C01815=1097.718,-43.728,-51.069,175.704,14.690,152.016
C01816=1097.724,-43.478,-51.082,175.706,14.691,152.016
C01817=1097.729,-43.229,-51.094,175.708,14.691,152.015
C01818=1097.736,-42.979,-51.106,175.710,14.692,152.015
C01819=1097.742,-42.730,-51.119,175.711,14.692,152.015
C01820=1097.748,-42.480,-51.130,175.713,14.693,152.015
C01821=1097.754,-42.230,-51.142,175.715,14.694,152.014
C01822=1097.759,-41.981,-51.154,175.717,14.695,152.014
C01823=1097.766,-41.731,-51.166,175.718,14.695,152.014
C01824=1097.771,-41.482,-51.179,175.720,14.696,152.014
C01825=1097.776,-41.232,-51.190,175.722,14.697,152.013
C01826=1097.783,-40.982,-51.202,175.724,14.697,152.013
C01827=1097.789,-40.732,-51.215,175.726,14.698,152.013
C01828=1097.795,-40.483,-51.226,175.728,14.699,152.012
C01829=1097.801,-40.234,-51.239,175.730,14.700,152.012
C01830=1097.807,-39.984,-51.252,175.732,14.700,152.012
C01831=1097.813,-39.735,-51.263,175.733,14.701,152.012
C01832=1097.819,-39.484,-51.275,175.735,14.702,152.011
C01833=1097.824,-39.234,-51.287,175.737,14.703,152.011
C01834=1097.831,-38.985,-51.299,175.739,14.703,152.011
C01835=1097.836,-38.736,-51.312,175.741,14.704,152.011
C01836=1097.842,-38.486,-51.324,175.743,14.705,152.010
C01837=1097.848,-38.236,-51.337,175.745,14.706,152.010
C01838=1097.854,-37.987,-51.348,175.747,14.706,152.010
C01839=1097.860,-37.737,-51.361,175.748,14.707,152.010
C01840=1097.866,-37.487,-51.373,175.750,14.708,152.009
C01841=1097.871,-37.238,-51.386,175.752,14.709,152.009
C01842=1097.877,-36.988,-51.397,175.754,14.709,152.009
C01843=1097.884,-36.738,-51.409,175.756,14.710,152.009
C01844=1097.889,-36.489,-51.422,175.758,14.711,152.008
C01845=1097.895,-36.239,-51.434,175.760,14.712,152.008
C01846=1097.901,-35.989,-51.447,175.762,14.712,152.008
C01847=1097.906,-35.740,-51.459,175.763,14.713,152.008
C01848=1097.912,-35.490,-51.471,175.765,14.714,152.007
C01849=1097.919,-35.240,-51.483,175.767,14.715,152.007
C01850=1097.924,-34.991,-51.496,175.769,14.715,152.007
C01851=1097.930,-34.741,-51.508,175.771,14.716,152.006
C01852=1097.936,-34.491,-51.521,175.773,14.717,152.006
C01853=1097.941,-34.242,-51.533,175.775,14.717,152.006
C01854=1097.947,-33.992,-51.545,175.777,14.718,152.006
C01855=1097.954,-33.743,-51.557,175.778,14.719,152.005
C01856=1097.960,-33.493,-51.570,175.780,14.720,152.005
C01857=1097.965,-33.244,-51.582,175.782,14.720,152.005
C01858=1097.971,-32.994,-51.595,175.784,14.721,152.005
C01859=1097.977,-32.727,-51.608,175.786,14.722,152.004
C01860=1097.984,-32.460,-51.622,175.788,14.723,152.004
C01861=1097.990,-32.192,-51.635,175.790,14.723,152.004
C01862=1097.996,-31.924,-51.648,175.792,14.725,152.004
C01863=1098.002,-31.674,-51.661,175.794,14.726,152.003
C01864=1098.008,-31.425,-51.673,175.796,14.726,152.003
C01865=1098.013,-31.175,-51.686,175.798,14.727,152.003
C01866=1098.020,-30.926,-51.698,175.800,14.728,152.003
C01867=1098.026,-30.677,-51.711,175.802,14.728,152.002
C01868=1098.032,-30.427,-51.723,175.804,14.729,152.002
C01869=1098.037,-30.178,-51.736,175.806,14.730,152.002
C01870=1098.043,-29.928,-51.748,175.807,14.731,152.001
C01871=1098.049,-29.678,-51.761,175.809,14.731,152.001
C01872=1098.055,-29.428,-51.773,175.812,14.732,152.001
C01873=1098.061,-29.178,-51.786,175.813,14.732,152.001
C01874=1098.066,-28.929,-51.799,175.815,14.733,152.000
C01875=1098.072,-28.680,-51.811,175.817,14.734,152.000
C01876=1098.078,-28.430,-51.824,175.819,14.735,152.000
C01877=1098.085,-28.180,-51.836,175.821,14.735,152.000
C01878=1098.091,-27.930,-51.848,175.823,14.736,151.999
C01879=1098.097,-27.681,-51.862,175.825,14.737,151.999
C01880=1098.102,-27.432,-51.874,175.827,14.738,151.999
C01881=1098.108,-27.182,-51.886,175.828,14.738,151.998
C01882=1098.114,-26.932,-51.899,175.830,14.739,151.998
C01883=1098.120,-26.682,-51.911,175.832,14.740,151.998
C01884=1098.126,-26.433,-51.925,175.834,14.741,151.998
C01885=1098.132,-26.184,-51.937,175.836,14.741,151.997
C01886=1098.137,-25.933,-51.950,175.838,14.742,151.997
C01887=1098.143,-25.684,-51.963,175.840,14.743,151.997
C01888=1098.149,-25.434,-51.976,175.842,14.744,151.997
C01889=1098.155,-25.184,-51.988,175.843,14.744,151.996
C01890=1098.160,-24.935,-52.001,175.845,14.745,151.996
C01891=1098.166,-24.685,-52.013,175.847,14.746,151.996
C01892=1098.172,-24.436,-52.026,175.850,14.747,151.996
C01893=1098.178,-24.186,-52.039,175.852,14.748,151.995
C01894=1098.184,-23.936,-52.052,175.854,14.749,151.995
C01895=1098.190,-23.688,-52.064,175.855,14.749,151.995
C01896=1098.195,-23.438,-52.078,175.857,14.750,151.995
C01897=1098.201,-23.188,-52.090,175.859,14.751,151.994
C01898=1098.207,-22.938,-52.103,175.861,14.752,151.994
C01899=1098.213,-22.689,-52.116,175.863,14.752,151.994
C01900=1098.219,-22.439,-52.129,175.865,14.753,151.993
C01901=1098.225,-22.189,-52.142,175.867,14.754,151.993
C01902=1098.230,-21.940,-52.154,175.869,14.755,151.993
C01903=1098.235,-21.690,-52.167,175.870,14.755,151.993
C01904=1098.242,-21.441,-52.180,175.872,14.756,151.992
C01905=1098.247,-21.191,-52.193,175.875,14.756,151.992
C01906=1098.254,-20.942,-52.206,175.876,14.757,151.992
C01907=1098.260,-20.692,-52.219,175.878,14.758,151.992
C01908=1098.266,-20.442,-52.231,175.881,14.759,151.991
C01909=1098.272,-20.193,-52.245,175.883,14.760,151.991
C01910=1098.276,-19.943,-52.257,175.885,14.761,151.991
C01911=1098.283,-19.694,-52.271,175.887,14.761,151.990
C01912=1098.288,-19.444,-52.283,175.888,14.762,151.990
C01913=1098.294,-19.194,-52.296,175.890,14.763,151.990
C01914=1098.301,-18.945,-52.309,175.892,14.764,151.990
C01915=1098.306,-18.695,-52.322,175.894,14.764,151.989
C01916=1098.312,-18.445,-52.336,175.896,14.765,151.989
C01917=1098.318,-18.195,-52.348,175.898,14.766,151.989
C01918=1098.324,-17.946,-52.361,175.900,14.767,151.989
C01919=1098.330,-17.696,-52.374,175.902,14.767,151.988
C01920=1098.335,-17.447,-52.388,175.904,14.768,151.988
C01921=1098.341,-17.197,-52.400,175.906,14.769,151.988
C01922=1098.347,-16.948,-52.413,175.908,14.770,151.987
C01923=1098.353,-16.680,-52.427,175.910,14.771,151.987
C01924=1098.359,-16.411,-52.441,175.912,14.771,151.987
C01925=1098.366,-16.143,-52.455,175.914,14.772,151.987
C01926=1098.373,-15.875,-52.469,175.917,14.773,151.986
C01927=1098.378,-15.625,-52.483,175.919,14.774,151.986
C01928=1098.384,-15.376,-52.496,175.921,14.774,151.986
C01929=1098.390,-15.126,-52.508,175.923,14.775,151.985
C01930=1098.397,-14.877,-52.522,175.924,14.776,151.985
C01931=1098.402,-14.626,-52.535,175.926,14.777,151.985
C01932=1098.408,-14.377,-52.548,175.928,14.777,151.985
C01933=1098.413,-14.128,-52.561,175.930,14.778,151.984
C01934=1098.419,-13.878,-52.574,175.932,14.779,151.984
C01935=1098.425,-13.629,-52.587,175.934,14.780,151.984
C01936=1098.430,-13.379,-52.601,175.936,14.781,151.984
C01937=1098.436,-13.130,-52.614,175.938,14.782,151.983
C01938=1098.441,-12.880,-52.627,175.940,14.783,151.983
C01939=1098.448,-12.630,-52.640,175.942,14.783,151.983
C01940=1098.454,-12.381,-52.654,175.944,14.784,151.982
C01941=1098.459,-12.131,-52.667,175.946,14.784,151.982
C01942=1098.465,-11.882,-52.680,175.948,14.785,151.982
C01943=1098.471,-11.632,-52.694,175.950,14.786,151.982
C01944=1098.477,-11.382,-52.706,175.952,14.787,151.981
C01945=1098.483,-11.133,-52.720,175.954,14.787,151.981
C01946=1098.488,-10.883,-52.734,175.956,14.789,151.981
C01947=1098.494,-10.633,-52.746,175.958,14.789,151.980
C01948=1098.500,-10.384,-52.760,175.960,14.790,151.980
C01949=1098.506,-10.135,-52.773,175.962,14.790,151.980
C01950=1098.511,-9.884,-52.786,175.964,14.791,151.980
C01951=1098.517,-9.635,-52.800,175.966,14.792,151.979
C01952=1098.524,-9.386,-52.813,175.968,14.793,151.979
C01953=1098.529,-9.136,-52.827,175.970,14.793,151.979
C01954=1098.535,-8.886,-52.839,175.972,14.795,151.978
C01955=1098.540,-8.637,-52.853,175.974,14.796,151.978
C01956=1098.547,-8.387,-52.866,175.976,14.796,151.978
C01957=1098.552,-8.138,-52.880,175.978,14.797,151.978
C01958=1098.558,-7.888,-52.893,175.980,14.797,151.977
C01959=1098.564,-7.638,-52.907,175.982,14.798,151.977
C01960=1098.570,-7.389,-52.920,175.984,14.799,151.977
C01961=1098.575,-7.140,-52.934,175.986,14.800,151.977
C01962=1098.581,-6.890,-52.947,175.989,14.801,151.976
C01963=1098.587,-6.640,-52.960,175.990,14.802,151.976
C01964=1098.593,-6.391,-52.974,175.993,14.802,151.976
C01965=1098.600,-6.141,-52.987,175.994,14.803,151.975
C01966=1098.605,-5.891,-53.001,175.996,14.803,151.975
C01967=1098.611,-5.642,-53.014,175.998,14.804,151.975
C01968=1098.617,-5.393,-53.028,176.000,14.805,151.975
C01969=1098.623,-5.143,-53.041,176.002,14.805,151.974
C01970=1098.628,-4.893,-53.055,176.005,14.807,151.974
C01971=1098.634,-4.643,-53.069,176.007,14.807,151.974
C01972=1098.640,-4.394,-53.082,176.009,14.808,151.973
C01973=1098.645,-4.145,-53.096,176.011,14.809,151.973
C01974=1098.652,-3.895,-53.109,176.012,14.810,151.973
C01975=1098.657,-3.646,-53.123,176.015,14.810,151.972
C01976=1098.664,-3.396,-53.136,176.017,14.811,151.972
C01977=1098.669,-3.146,-53.150,176.018,14.811,151.972
C01978=1098.676,-2.897,-53.164,176.021,14.813,151.972
C01979=1098.681,-2.647,-53.177,176.023,14.813,151.971
C01980=1098.686,-2.397,-53.191,176.025,14.814,151.971
C01981=1098.692,-2.148,-53.204,176.027,14.814,151.971
C01982=1098.698,-1.898,-53.218,176.029,14.815,151.970
C01983=1098.703,-1.649,-53.232,176.031,14.816,151.970
C01984=1098.709,-1.399,-53.245,176.033,14.817,151.970
C01985=1098.715,-1.150,-53.259,176.035,14.818,151.970
C01986=1098.721,-0.900,-53.273,176.037,14.819,151.969
C01987=1098.726,-0.630,-53.287,176.039,14.820,151.969
C01988=1098.733,-0.360,-53.302,176.042,14.820,151.969
C01989=1098.739,-0.091,-53.318,176.044,14.821,151.968
C01990=1098.745,0.179,-53.332,176.046,14.822,151.968
C01991=1098.751,0.429,-53.346,176.048,14.823,151.968
C01992=1098.756,0.678,-53.360,176.051,14.824,151.967
C01993=1098.762,0.927,-53.373,176.052,14.824,151.967
C01994=1098.769,1.178,-53.387,176.054,14.825,151.967
C01995=1098.774,1.427,-53.401,176.056,14.826,151.967
C01996=1098.779,1.677,-53.415,176.058,14.827,151.966
C01997=1098.786,1.926,-53.428,176.060,14.827,151.966
C01998=1098.791,2.176,-53.442,176.063,14.828,151.966
C01999=1098.797,2.425,-53.456,176.065,14.829,151.965
C02000=1098.802,2.675,-53.470,176.067,14.830,151.965
C02001=1098.808,2.924,-53.484,176.069,14.830,151.965
C02002=1098.814,3.174,-53.498,176.071,14.831,151.964
C02003=1098.820,3.423,-53.512,176.073,14.832,151.964
C02004=1098.826,3.673,-53.526,176.075,14.833,151.964
C02005=1098.831,3.922,-53.540,176.077,14.834,151.964
C02006=1098.837,4.172,-53.554,176.079,14.834,151.963
C02007=1098.843,4.421,-53.567,176.081,14.835,151.963
C02008=1098.849,4.672,-53.581,176.083,14.835,151.963
C02009=1098.854,4.921,-53.595,176.085,14.836,151.962
C02010=1098.860,5.170,-53.610,176.088,14.838,151.962
C02011=1098.866,5.420,-53.624,176.090,14.838,151.962
C02012=1098.872,5.669,-53.637,176.092,14.839,151.961
C02013=1098.878,5.919,-53.651,176.094,14.839,151.961
C02014=1098.883,6.169,-53.665,176.096,14.840,151.961
C02015=1098.889,6.418,-53.679,176.098,14.840,151.961
C02016=1098.895,6.667,-53.693,176.100,14.842,151.960
C02017=1098.900,6.917,-53.707,176.102,14.842,151.960
C02018=1098.907,7.167,-53.721,176.104,14.843,151.960
C02019=1098.912,7.416,-53.735,176.106,14.844,151.959
C02020=1098.918,7.665,-53.749,176.108,14.844,151.959
C02021=1098.924,7.915,-53.763,176.111,14.845,151.959
C02022=1098.930,8.165,-53.777,176.113,14.846,151.958
C02023=1098.935,8.415,-53.791,176.115,14.847,151.958
C02024=1098.941,8.664,-53.806,176.117,14.847,151.958
C02025=1098.947,8.913,-53.819,176.119,14.848,151.957
C02026=1098.953,9.163,-53.833,176.122,14.849,151.957
C02027=1098.959,9.412,-53.848,176.123,14.850,151.957
C02028=1098.965,9.662,-53.862,176.126,14.850,151.956
C02029=1098.970,9.911,-53.876,176.127,14.851,151.956
C02030=1098.976,10.161,-53.891,176.129,14.852,151.956
C02031=1098.982,10.411,-53.904,176.132,14.852,151.956
C02032=1098.987,10.660,-53.918,176.134,14.853,151.955
C02033=1098.994,10.910,-53.933,176.136,14.854,151.955
C02034=1098.999,11.159,-53.947,176.138,14.854,151.955
C02035=1099.005,11.409,-53.960,176.140,14.855,151.954
C02036=1099.012,11.658,-53.975,176.142,14.855,151.954
C02037=1099.017,11.908,-53.989,176.145,14.857,151.954
C02038=1099.023,12.158,-54.003,176.147,14.857,151.953
C02039=1099.029,12.407,-54.018,176.149,14.858,151.953
C02040=1099.035,12.657,-54.032,176.151,14.858,151.953
C02041=1099.040,12.906,-54.046,176.153,14.859,151.952
C02042=1099.046,13.155,-54.060,176.156,14.860,151.952
C02043=1099.052,13.405,-54.075,176.158,14.861,151.952
C02044=1099.058,13.655,-54.089,176.160,14.861,151.951
C02045=1099.064,13.905,-54.103,176.162,14.862,151.951
C02046=1099.070,14.154,-54.118,176.164,14.862,151.951
C02047=1099.075,14.403,-54.132,176.167,14.864,151.950
C02048=1099.081,14.652,-54.146,176.168,14.864,151.950
C02049=1099.087,14.903,-54.161,176.171,14.865,151.950
C02050=1099.093,15.152,-54.175,176.173,14.865,151.949
C02051=1099.099,15.424,-54.190,176.175,14.866,151.949
C02052=1099.105,15.695,-54.206,176.177,14.867,151.949
C02053=1099.111,15.968,-54.222,176.180,14.868,151.948
C02054=1099.118,16.239,-54.238,176.182,14.869,151.948
C02055=1099.123,16.489,-54.252,176.184,14.869,151.948
C02056=1099.130,16.738,-54.266,176.186,14.870,151.947
C02057=1099.135,16.987,-54.281,176.189,14.871,151.947
C02058=1099.140,17.237,-54.296,176.191,14.871,151.947
C02059=1099.147,17.487,-54.310,176.193,14.872,151.946
C02060=1099.152,17.736,-54.324,176.195,14.873,151.946
C02061=1099.158,17.985,-54.339,176.198,14.874,151.946
C02062=1099.164,18.236,-54.353,176.200,14.875,151.945
C02063=1099.170,18.485,-54.368,176.202,14.875,151.945
C02064=1099.176,18.734,-54.383,176.204,14.876,151.945
C02065=1099.181,18.984,-54.397,176.206,14.876,151.944
C02066=1099.187,19.233,-54.412,176.209,14.877,151.944
C02067=1099.193,19.483,-54.426,176.210,14.878,151.944
C02068=1099.198,19.732,-54.441,176.213,14.878,151.943
C02069=1099.205,19.982,-54.455,176.215,14.879,151.943
C02070=1099.210,20.232,-54.469,176.218,14.880,151.943
C02071=1099.215,20.481,-54.484,176.219,14.881,151.942
C02072=1099.222,20.730,-54.499,176.222,14.881,151.942
C02073=1099.227,20.980,-54.513,176.223,14.882,151.942
C02074=1099.233,21.229,-54.528,176.226,14.883,151.941
C02075=1099.239,21.479,-54.543,176.228,14.883,151.941
C02076=1099.244,21.729,-54.557,176.230,14.884,151.941
C02077=1099.251,21.978,-54.572,176.232,14.884,151.940
C02078=1099.256,22.227,-54.587,176.234,14.885,151.940
C02079=1099.261,22.477,-54.601,176.237,14.886,151.940
C02080=1099.267,22.727,-54.616,176.239,14.887,151.939
C02081=1099.273,22.976,-54.631,176.241,14.887,151.939
C02082=1099.279,23.226,-54.645,176.243,14.888,151.939
C02083=1099.284,23.475,-54.660,176.246,14.889,151.938
C02084=1099.290,23.724,-54.675,176.248,14.890,151.938
C02085=1099.296,23.974,-54.690,176.250,14.890,151.938
C02086=1099.301,24.224,-54.704,176.252,14.891,151.937
C02087=1099.308,24.473,-54.719,176.255,14.891,151.937
C02088=1099.313,24.722,-54.734,176.257,14.892,151.937
C02089=1099.320,24.972,-54.749,176.259,14.893,151.936
C02090=1099.325,25.221,-54.764,176.261,14.893,151.936
C02091=1099.331,25.472,-54.778,176.264,14.894,151.935
C02092=1099.337,25.720,-54.793,176.266,14.894,151.935
C02093=1099.342,25.970,-54.808,176.268,14.895,151.935
C02094=1099.348,26.219,-54.823,176.270,14.896,151.934
C02095=1099.354,26.469,-54.838,176.273,14.897,151.934
C02096=1099.360,26.718,-54.853,176.275,14.897,151.934
C02097=1099.365,26.968,-54.867,176.277,14.898,151.933
C02098=1099.371,27.218,-54.882,176.279,14.898,151.933
C02099=1099.376,27.467,-54.897,176.282,14.900,151.933
C02100=1099.383,27.716,-54.912,176.284,14.900,151.932
C02101=1099.388,27.966,-54.927,176.286,14.900,151.932
C02102=1099.394,28.215,-54.942,176.288,14.901,151.932
C02103=1099.400,28.464,-54.957,176.291,14.902,151.931
C02104=1099.406,28.714,-54.972,176.293,14.903,151.931
C02105=1099.411,28.963,-54.987,176.295,14.903,151.931
C02106=1099.417,29.213,-55.002,176.298,14.904,151.930
C02107=1099.423,29.463,-55.016,176.300,14.905,151.930
C02108=1099.428,29.713,-55.032,176.302,14.905,151.929
C02109=1099.434,29.962,-55.046,176.304,14.906,151.929
C02110=1099.440,30.212,-55.062,176.307,14.906,151.929
C02111=1099.445,30.461,-55.076,176.309,14.907,151.928
C02112=1099.451,30.711,-55.092,176.311,14.908,151.928
C02113=1099.457,30.960,-55.106,176.313,14.908,151.928
C02114=1099.463,31.210,-55.122,176.316,14.909,151.927
C02115=1099.469,31.483,-55.138,176.318,14.910,151.927
C02116=1099.475,31.756,-55.155,176.321,14.910,151.926
C02117=1099.482,32.029,-55.171,176.323,14.911,151.926
C02118=1099.487,32.303,-55.188,176.326,14.912,151.926
C02119=1099.494,32.552,-55.203,176.328,14.912,151.925
C02120=1099.499,32.801,-55.218,176.330,14.913,151.925
C02121=1099.505,33.051,-55.233,176.333,14.914,151.925
C02122=1099.510,33.300,-55.249,176.335,14.914,151.924
C02123=1099.517,33.549,-55.264,176.337,14.915,151.924
C02124=1099.522,33.799,-55.279,176.339,14.915,151.924
C02125=1099.528,34.048,-55.294,176.342,14.916,151.923
C02126=1099.534,34.298,-55.309,176.344,14.917,151.923
C02127=1099.540,34.547,-55.324,176.346,14.917,151.922
C02128=1099.545,34.797,-55.340,176.349,14.918,151.922
C02129=1099.550,35.047,-55.355,176.351,14.919,151.922
C02130=1099.557,35.296,-55.370,176.353,14.919,151.921
C02131=1099.562,35.546,-55.385,176.355,14.920,151.921
C02132=1099.569,35.794,-55.401,176.358,14.920,151.920
C02133=1099.574,36.044,-55.416,176.360,14.921,151.920
C02134=1099.580,36.293,-55.431,176.362,14.922,151.920
C02135=1099.586,36.543,-55.446,176.365,14.922,151.919
C02136=1099.591,36.793,-55.462,176.367,14.923,151.919
C02137=1099.597,37.042,-55.476,176.369,14.924,151.919
C02138=1099.603,37.292,-55.493,176.372,14.924,151.918
C02139=1099.609,37.541,-55.508,176.375,14.925,151.918
C02140=1099.614,37.791,-55.523,176.377,14.925,151.917
C02141=1099.620,38.041,-55.538,176.379,14.926,151.917
C02142=1099.625,38.289,-55.554,176.382,14.927,151.917
C02143=1099.632,38.539,-55.569,176.384,14.927,151.916
C02144=1099.637,38.789,-55.585,176.386,14.927,151.916
C02145=1099.642,39.038,-55.600,176.388,14.928,151.916
C02146=1099.649,39.287,-55.615,176.391,14.929,151.915
C02147=1099.654,39.536,-55.631,176.393,14.929,151.915
C02148=1099.660,39.786,-55.646,176.395,14.930,151.914
C02149=1099.665,40.036,-55.662,176.398,14.931,151.914
C02150=1099.672,40.285,-55.677,176.400,14.931,151.914
C02151=1099.677,40.535,-55.693,176.402,14.931,151.913
C02152=1099.683,40.785,-55.708,176.405,14.932,151.913
C02153=1099.688,41.033,-55.724,176.407,14.933,151.913
C02154=1099.695,41.283,-55.739,176.409,14.933,151.912
C02155=1099.700,41.533,-55.754,176.412,14.934,151.912
C02156=1099.706,41.781,-55.770,176.414,14.935,151.911
C02157=1099.711,42.031,-55.786,176.417,14.935,151.911
C02158=1099.717,42.281,-55.801,176.418,14.936,151.911
C02159=1099.723,42.530,-55.817,176.421,14.937,151.910
C02160=1099.729,42.780,-55.832,176.424,14.937,151.910
C02161=1099.734,43.030,-55.848,176.426,14.937,151.909
C02162=1099.740,43.278,-55.864,176.429,14.938,151.909
C02163=1099.745,43.528,-55.879,176.431,14.938,151.908
C02164=1099.752,43.777,-55.895,176.433,14.939,151.908
C02165=1099.757,44.027,-55.910,176.436,14.940,151.908
C02166=1099.763,44.277,-55.926,176.438,14.940,151.907
C02167=1099.769,44.526,-55.942,176.440,14.941,151.907
C02168=1099.774,44.775,-55.957,176.443,14.942,151.906
C02169=1099.780,45.025,-55.973,176.445,14.942,151.906
C02170=1099.785,45.275,-55.989,176.447,14.943,151.906
C02171=1099.791,45.523,-56.005,176.450,14.944,151.905
C02172=1099.796,45.773,-56.020,176.452,14.944,151.905
C02173=1099.802,46.022,-56.037,176.454,14.944,151.905
C02174=1099.807,46.272,-56.052,176.457,14.945,151.904
C02175=1099.813,46.521,-56.068,176.459,14.946,151.904
C02176=1099.819,46.771,-56.084,176.461,14.946,151.903
C02177=1099.824,47.020,-56.099,176.464,14.947,151.903
C02178=1099.830,47.270,-56.115,176.467,14.947,151.903
C02179=1099.836,47.543,-56.133,176.470,14.948,151.902
C02180=1099.842,47.816,-56.150,176.472,14.949,151.902
C02181=1099.848,48.090,-56.167,176.475,14.950,151.901
C02182=1099.854,48.363,-56.184,176.477,14.950,151.901
C02183=1099.860,48.612,-56.200,176.480,14.951,151.900
C02184=1099.866,48.862,-56.216,176.482,14.951,151.900
C02185=1099.872,49.111,-56.232,176.484,14.951,151.900
C02186=1099.877,49.360,-56.248,176.487,14.952,151.899
C02187=1099.883,49.610,-56.263,176.489,14.953,151.899
C02188=1099.889,49.859,-56.280,176.492,14.953,151.898
C02189=1099.894,50.109,-56.295,176.495,14.954,151.898
C02190=1099.900,50.358,-56.311,176.497,14.954,151.897
C02191=1099.906,50.607,-56.327,176.499,14.954,151.897
C02192=1099.911,50.857,-56.343,176.502,14.955,151.897
C02193=1099.917,51.107,-56.359,176.504,14.956,151.896
C02194=1099.923,51.356,-56.375,176.506,14.956,151.896
C02195=1099.928,51.606,-56.391,176.509,14.957,151.895
C02196=1099.934,51.855,-56.407,176.511,14.957,151.895
C02197=1099.940,52.104,-56.424,176.514,14.957,151.894
C02198=1099.945,52.354,-56.439,176.517,14.958,151.894
C02199=1099.951,52.604,-56.455,176.519,14.959,151.894
C02200=1099.957,52.852,-56.471,176.521,14.959,151.893
C02201=1099.962,53.102,-56.488,176.524,14.960,151.893
C02202=1099.968,53.352,-56.503,176.526,14.960,151.892
C02203=1099.974,53.601,-56.519,176.528,14.960,151.892
C02204=1099.980,53.850,-56.536,176.531,14.961,151.891
C02205=1099.986,54.100,-56.552,176.533,14.962,151.891
C02206=1099.991,54.349,-56.567,176.536,14.962,151.891
C02207=1099.996,54.599,-56.584,176.539,14.963,151.890
C02208=1100.002,54.848,-56.600,176.541,14.963,151.890
C02209=1100.008,55.097,-56.616,176.543,14.964,151.889
C02210=1100.014,55.347,-56.633,176.546,14.964,151.889
C02211=1100.020,55.597,-56.648,176.548,14.965,151.889
C02212=1100.026,55.846,-56.665,176.551,14.965,151.888
C02213=1100.031,56.095,-56.680,176.554,14.965,151.887
C02214=1100.037,56.344,-56.697,176.556,14.966,151.887
C02215=1100.042,56.594,-56.714,176.559,14.967,151.887
C02216=1100.048,56.843,-56.730,176.561,14.967,151.886
C02217=1100.054,57.093,-56.745,176.563,14.967,151.886
C02218=1100.060,57.342,-56.762,176.566,14.968,151.885
C02219=1100.066,57.592,-56.778,176.569,14.968,151.885
C02220=1100.072,57.841,-56.794,176.571,14.968,151.884
C02221=1100.077,58.091,-56.811,176.574,14.969,151.884
C02222=1100.083,58.340,-56.827,176.576,14.970,151.884
C02223=1100.089,58.589,-56.843,176.578,14.970,151.883
C02224=1100.095,58.839,-56.860,176.581,14.970,151.882
C02225=1100.100,59.087,-56.876,176.584,14.971,151.882
C02226=1100.106,59.337,-56.892,176.586,14.971,151.882
C02227=1100.111,59.586,-56.909,176.589,14.972,151.881
C02228=1100.117,59.836,-56.925,176.591,14.972,151.881
C02229=1100.123,60.085,-56.941,176.594,14.973,151.880
C02230=1100.129,60.334,-56.957,176.596,14.973,151.880
C02231=1100.135,60.584,-56.974,176.599,14.973,151.879
C02232=1100.140,60.833,-56.991,176.602,14.974,151.879
C02233=1100.146,61.083,-57.007,176.604,14.974,151.878
C02234=1100.152,61.332,-57.023,176.606,14.974,151.878
C02235=1100.158,61.581,-57.039,176.609,14.975,151.877
C02236=1100.163,61.831,-57.056,176.612,14.975,151.877
C02237=1100.169,62.080,-57.072,176.614,14.975,151.877
C02238=1100.175,62.330,-57.089,176.617,14.976,151.876
C02239=1100.181,62.579,-57.105,176.619,14.976,151.875
C02240=1100.186,62.829,-57.122,176.622,14.977,151.875
C02241=1100.192,63.078,-57.138,176.625,14.977,151.875
C02242=1100.198,63.327,-57.154,176.627,14.977,151.874
C02243=1100.205,63.600,-57.173,176.630,14.978,151.874
C02244=1100.211,63.874,-57.191,176.632,14.978,151.873
C02245=1100.218,64.147,-57.209,176.635,14.979,151.873
C02246=1100.224,64.420,-57.226,176.639,14.979,151.872
C02247=1100.230,64.668,-57.243,176.641,14.980,151.872
C02248=1100.235,64.918,-57.260,176.643,14.980,151.871
C02249=1100.241,65.167,-57.276,176.646,14.981,151.871
C02250=1100.246,65.417,-57.293,176.649,14.981,151.870
C02251=1100.252,65.666,-57.310,176.652,14.982,151.870
C02252=1100.257,65.916,-57.326,176.654,14.982,151.869
C02253=1100.264,66.166,-57.343,176.656,14.982,151.869
C02254=1100.270,66.415,-57.360,176.659,14.983,151.868
C02255=1100.275,66.665,-57.377,176.662,14.983,151.868
C02256=1100.281,66.914,-57.393,176.664,14.983,151.867
C02257=1100.287,67.164,-57.410,176.667,14.983,151.867
C02258=1100.293,67.412,-57.427,176.669,14.984,151.866
C02259=1100.298,67.662,-57.444,176.672,14.985,151.866
C02260=1100.304,67.911,-57.460,176.675,14.985,151.865
C02261=1100.309,68.161,-57.477,176.677,14.985,151.865
C02262=1100.315,68.410,-57.494,176.680,14.986,151.864
C02263=1100.321,68.659,-57.511,176.682,14.986,151.864
C02264=1100.327,68.909,-57.527,176.685,14.987,151.863
C02265=1100.332,69.158,-57.544,176.688,14.986,151.863
C02266=1100.338,69.407,-57.561,176.690,14.987,151.862
C02267=1100.343,69.657,-57.578,176.693,14.987,151.862
C02268=1100.349,69.906,-57.594,176.696,14.987,151.861
C02269=1100.355,70.155,-57.612,176.698,14.988,151.861
C02270=1100.361,70.404,-57.628,176.701,14.988,151.860
C02271=1100.366,70.654,-57.645,176.703,14.989,151.860
C02272=1100.372,70.904,-57.663,176.706,14.989,151.859
C02273=1100.378,71.153,-57.679,176.709,14.989,151.859
C02274=1100.383,71.403,-57.696,176.711,14.989,151.858
C02275=1100.389,71.652,-57.713,176.714,14.990,151.858
C02276=1100.395,71.901,-57.729,176.717,14.990,151.857
C02277=1100.400,72.150,-57.747,176.720,14.991,151.857
C02278=1100.406,72.400,-57.763,176.722,14.991,151.856
C02279=1100.411,72.649,-57.780,176.724,14.991,151.856
C02280=1100.418,72.898,-57.797,176.728,14.992,151.855
C02281=1100.423,73.148,-57.814,176.730,14.992,151.855
C02282=1100.428,73.397,-57.832,176.733,14.992,151.854
C02283=1100.435,73.647,-57.848,176.735,14.993,151.854
C02284=1100.440,73.896,-57.866,176.738,14.993,151.853
C02285=1100.446,74.145,-57.883,176.741,14.993,151.853
C02286=1100.452,74.394,-57.900,176.743,14.993,151.852
C02287=1100.457,74.644,-57.916,176.746,14.994,151.852
C02288=1100.463,74.893,-57.934,176.749,14.994,151.851
C02289=1100.469,75.142,-57.950,176.751,14.994,151.851
C02290=1100.475,75.392,-57.968,176.754,14.995,151.850
C02291=1100.480,75.642,-57.985,176.756,14.995,151.850
C02292=1100.486,75.890,-58.002,176.760,14.996,151.849
C02293=1100.491,76.140,-58.019,176.762,14.996,151.849
C02294=1100.497,76.389,-58.036,176.765,14.996,151.848
C02295=1100.502,76.639,-58.053,176.768,14.996,151.848
C02296=1100.509,76.888,-58.071,176.770,14.996,151.847
C02297=1100.514,77.137,-58.088,176.773,14.997,151.847
C02298=1100.520,77.387,-58.105,176.775,14.997,151.846
C02299=1100.526,77.636,-58.122,176.778,14.998,151.846
C02300=1100.531,77.885,-58.139,176.781,14.998,151.845
C02301=1100.537,78.135,-58.157,176.783,14.998,151.845
C02302=1100.543,78.384,-58.174,176.786,14.999,151.844
C02303=1100.548,78.634,-58.191,176.789,14.998,151.843
C02304=1100.554,78.882,-58.208,176.792,14.999,151.843
C02305=1100.559,79.132,-58.225,176.794,14.999,151.842
C02306=1100.566,79.382,-58.243,176.797,14.999,151.842
C02307=1100.572,79.655,-58.262,176.800,15.000,151.841
C02308=1100.577,79.927,-58.280,176.803,15.000,151.841
C02309=1100.584,80.200,-58.300,176.806,15.000,151.840
C02310=1100.590,80.473,-58.319,176.809,15.000,151.840
C02311=1100.596,80.723,-58.337,176.811,15.001,151.839
C02312=1100.601,80.973,-58.354,176.815,15.001,151.839
C02313=1100.607,81.221,-58.371,176.817,15.001,151.838
C02314=1100.613,81.470,-58.388,176.820,15.002,151.837
C02315=1100.618,81.720,-58.405,176.823,15.002,151.837
C02316=1100.624,81.970,-58.423,176.826,15.002,151.836
C02317=1100.630,82.219,-58.441,176.828,15.003,151.836
C02318=1100.635,82.468,-58.458,176.831,15.002,151.835
C02319=1100.641,82.717,-58.476,176.834,15.003,151.835
C02320=1100.646,82.967,-58.493,176.836,15.003,151.834
C02321=1100.652,83.216,-58.511,176.839,15.004,151.834
C02322=1100.658,83.465,-58.528,176.842,15.004,151.833
C02323=1100.663,83.714,-58.546,176.845,15.004,151.833
C02324=1100.669,83.964,-58.564,176.848,15.004,151.832
C02325=1100.674,84.214,-58.580,176.850,15.004,151.831
C02326=1100.680,84.463,-58.598,176.853,15.005,151.831
C02327=1100.686,84.713,-58.616,176.856,15.005,151.830
C02328=1100.692,84.962,-58.634,176.859,15.005,151.830
C02329=1100.698,85.210,-58.650,176.861,15.005,151.829
C02330=1100.703,85.459,-58.668,176.865,15.005,151.829
C02331=1100.709,85.709,-58.686,176.867,15.006,151.828
C02332=1100.715,85.958,-58.704,176.869,15.006,151.828
C02333=1100.720,86.208,-58.720,176.873,15.006,151.827
C02334=1100.726,86.457,-58.738,176.875,15.006,151.826
C02335=1100.732,86.707,-58.756,176.878,15.006,151.826
C02336=1100.737,86.956,-58.773,176.881,15.006,151.825
C02337=1100.743,87.205,-58.791,176.884,15.007,151.825
C02338=1100.749,87.454,-58.809,176.887,15.007,151.824
C02339=1100.754,87.703,-58.827,176.889,15.007,151.824
C02340=1100.761,87.953,-58.844,176.892,15.007,151.823
C02341=1100.765,88.202,-58.863,176.895,15.007,151.823
C02342=1100.771,88.452,-58.881,176.898,15.008,151.822
C02343=1100.777,88.701,-58.898,176.900,15.008,151.821
C02344=1100.783,88.950,-58.916,176.904,15.008,151.821
C02345=1100.789,89.200,-58.934,176.906,15.008,151.820
C02346=1100.794,89.449,-58.951,176.909,15.008,151.820
C02347=1100.800,89.698,-58.969,176.912,15.008,151.819
C02348=1100.806,89.948,-58.987,176.914,15.008,151.818
C02349=1100.811,90.197,-59.004,176.918,15.009,151.818
C02350=1100.818,90.446,-59.023,176.920,15.009,151.817
C02351=1100.823,90.695,-59.040,176.923,15.009,151.817
C02352=1100.829,90.945,-59.058,176.926,15.009,151.816
C02353=1100.835,91.194,-59.076,176.929,15.009,151.816
C02354=1100.840,91.443,-59.094,176.932,15.009,151.815
C02355=1100.846,91.693,-59.112,176.934,15.009,151.814
C02356=1100.851,91.942,-59.130,176.937,15.010,151.814
C02357=1100.857,92.191,-59.147,176.940,15.010,151.813
C02358=1100.863,92.441,-59.165,176.943,15.010,151.813
C02359=1100.868,92.689,-59.184,176.946,15.010,151.812
C02360=1100.874,92.939,-59.202,176.949,15.010,151.811
C02361=1100.880,93.188,-59.220,176.952,15.010,151.811
C02362=1100.885,93.437,-59.237,176.955,15.011,151.810
C02363=1100.891,93.687,-59.256,176.957,15.011,151.810
C02364=1100.896,93.936,-59.273,176.960,15.011,151.809
C02365=1100.903,94.186,-59.292,176.963,15.011,151.809
C02366=1100.908,94.435,-59.309,176.966,15.011,151.808
C02367=1100.913,94.684,-59.328,176.969,15.011,151.807
C02368=1100.919,94.934,-59.345,176.971,15.011,151.807
C02369=1100.925,95.182,-59.364,176.975,15.011,151.806
C02370=1100.931,95.432,-59.382,176.977,15.011,151.805
C02371=1100.937,95.705,-59.402,176.981,15.012,151.805
C02372=1100.943,95.978,-59.421,176.984,15.012,151.804
C02373=1100.949,96.251,-59.441,176.987,15.012,151.804
C02374=1100.955,96.524,-59.461,176.990,15.012,151.803
C02375=1100.961,96.774,-59.479,176.993,15.012,151.802
C02376=1100.966,97.022,-59.498,176.996,15.012,151.802
C02377=1100.973,97.272,-59.516,176.999,15.012,151.801
C02378=1100.978,97.521,-59.533,177.002,15.012,151.800
C02379=1100.983,97.770,-59.552,177.004,15.012,151.800
C02380=1100.989,98.020,-59.570,177.008,15.013,151.799
C02381=1100.995,98.269,-59.588,177.011,15.012,151.799
C02382=1101.001,98.518,-59.607,177.014,15.013,151.798
C02383=1101.007,98.768,-59.625,177.016,15.012,151.797
C02384=1101.012,99.016,-59.643,177.019,15.012,151.797
C02385=1101.018,99.266,-59.662,177.022,15.013,151.796
C02386=1101.023,99.515,-59.679,177.025,15.012,151.795
C02387=1101.030,99.764,-59.698,177.028,15.013,151.795
C02388=1101.035,100.014,-59.716,177.031,15.013,151.794
C02389=1101.041,100.263,-59.735,177.034,15.013,151.794
C02390=1101.047,100.512,-59.752,177.037,15.013,151.793
C02391=1101.052,100.761,-59.772,177.040,15.013,151.792
C02392=1101.058,101.010,-59.789,177.042,15.013,151.792
C02393=1101.063,101.260,-59.808,177.046,15.013,151.791
C02394=1101.070,101.510,-59.826,177.049,15.013,151.790
C02395=1101.075,101.758,-59.845,177.052,15.013,151.790
C02396=1101.081,102.008,-59.863,177.054,15.013,151.789
C02397=1101.086,102.257,-59.882,177.057,15.013,151.789
C02398=1101.092,102.507,-59.900,177.060,15.013,151.788
C02399=1101.097,102.755,-59.919,177.063,15.013,151.787
C02400=1101.103,103.005,-59.937,177.067,15.013,151.787
C02401=1101.108,103.254,-59.956,177.069,15.013,151.786
C02402=1101.114,103.504,-59.974,177.072,15.013,151.785
C02403=1101.119,103.752,-59.992,177.075,15.013,151.785
C02404=1101.126,104.002,-60.010,177.078,15.013,151.784
C02405=1101.131,104.251,-60.030,177.081,15.013,151.784
C02406=1101.136,104.500,-60.048,177.084,15.014,151.783
C02407=1101.142,104.750,-60.066,177.087,15.013,151.782
C02408=1101.148,104.999,-60.085,177.090,15.014,151.782
C02409=1101.154,105.248,-60.104,177.093,15.013,151.781
C02410=1101.159,105.498,-60.122,177.096,15.014,151.780
C02411=1101.165,105.746,-60.141,177.099,15.014,151.780
C02412=1101.171,105.996,-60.159,177.102,15.014,151.779
C02413=1101.176,106.245,-60.178,177.105,15.013,151.778
C02414=1101.182,106.494,-60.197,177.108,15.013,151.778
C02415=1101.188,106.744,-60.216,177.111,15.013,151.777
C02416=1101.193,106.993,-60.234,177.113,15.013,151.776
C02417=1101.199,107.242,-60.253,177.117,15.013,151.776
C02418=1101.205,107.491,-60.272,177.120,15.013,151.775
C02419=1101.210,107.741,-60.290,177.123,15.013,151.774
C02420=1101.216,107.990,-60.309,177.126,15.013,151.774
C02421=1101.222,108.239,-60.328,177.129,15.013,151.773
C02422=1101.227,108.488,-60.346,177.132,15.013,151.773
C02423=1101.233,108.738,-60.365,177.135,15.013,151.772
C02424=1101.239,108.987,-60.384,177.138,15.013,151.771
C02425=1101.244,109.236,-60.402,177.141,15.013,151.770
C02426=1101.250,109.485,-60.422,177.144,15.013,151.770
C02427=1101.256,109.734,-60.440,177.147,15.013,151.769
C02428=1101.261,109.984,-60.459,177.150,15.013,151.769
C02429=1101.267,110.233,-60.478,177.154,15.013,151.768
C02430=1101.273,110.482,-60.496,177.156,15.012,151.767
C02431=1101.278,110.731,-60.515,177.160,15.013,151.766
C02432=1101.284,110.980,-60.535,177.162,15.012,151.766
C02433=1101.290,111.229,-60.553,177.166,15.013,151.765
C02434=1101.296,111.479,-60.572,177.169,15.012,151.764
C02435=1101.302,111.752,-60.593,177.172,15.012,151.764
C02436=1101.308,112.025,-60.613,177.175,15.012,151.763
C02437=1101.315,112.298,-60.635,177.179,15.012,151.762
C02438=1101.320,112.571,-60.655,177.182,15.012,151.761
C02439=1101.326,112.821,-60.674,177.185,15.012,151.761
C02440=1101.332,113.070,-60.693,177.188,15.012,151.760
C02441=1101.338,113.319,-60.712,177.191,15.011,151.759
C02442=1101.343,113.568,-60.731,177.194,15.012,151.759
C02443=1101.349,113.817,-60.750,177.197,15.011,151.758
C02444=1101.355,114.067,-60.769,177.201,15.011,151.757
C02445=1101.360,114.316,-60.789,177.203,15.011,151.757
C02446=1101.366,114.565,-60.807,177.207,15.011,151.756
C02447=1101.372,114.814,-60.826,177.209,15.011,151.755
C02448=1101.377,115.063,-60.845,177.213,15.011,151.755
C02449=1101.383,115.312,-60.864,177.216,15.011,151.754
C02450=1101.388,115.562,-60.883,177.219,15.011,151.753
C02451=1101.394,115.811,-60.903,177.222,15.011,151.753
C02452=1101.400,116.060,-60.922,177.225,15.011,151.752
C02453=1101.405,116.309,-60.941,177.228,15.011,151.751
C02454=1101.410,116.559,-60.960,177.231,15.011,151.750
C02455=1101.416,116.808,-60.979,177.234,15.010,151.750
C02456=1101.422,117.057,-60.999,177.238,15.011,151.749
C02457=1101.427,117.306,-61.018,177.240,15.010,151.748
C02458=1101.433,117.555,-61.037,177.244,15.010,151.748
C02459=1101.439,117.804,-61.057,177.246,15.010,151.747
C02460=1101.444,118.054,-61.076,177.250,15.010,151.746
C02461=1101.449,118.303,-61.095,177.253,15.010,151.746
C02462=1101.455,118.552,-61.114,177.256,15.010,151.745
C02463=1101.461,118.801,-61.133,177.259,15.009,151.744
C02464=1101.467,119.050,-61.153,177.262,15.010,151.743
C02465=1101.472,119.300,-61.172,177.265,15.009,151.743
C02466=1101.477,119.548,-61.191,177.269,15.009,151.742
C02467=1101.483,119.798,-61.211,177.271,15.009,151.741
C02468=1101.489,120.047,-61.230,177.275,15.009,151.741
C02469=1101.495,120.296,-61.250,177.278,15.008,151.740
C02470=1101.500,120.546,-61.269,177.281,15.009,151.739
C02471=1101.506,120.795,-61.288,177.284,15.008,151.738
C02472=1101.511,121.044,-61.307,177.288,15.008,151.738
C02473=1101.517,121.293,-61.327,177.290,15.008,151.737
C02474=1101.523,121.542,-61.346,177.294,15.008,151.736
C02475=1101.529,121.791,-61.366,177.297,15.008,151.736
C02476=1101.534,122.041,-61.385,177.300,15.008,151.735
C02477=1101.540,122.290,-61.405,177.303,15.007,151.734
C02478=1101.545,122.539,-61.425,177.307,15.007,151.733
C02479=1101.551,122.789,-61.444,177.309,15.007,151.733
C02480=1101.556,123.037,-61.463,177.313,15.007,151.732
C02481=1101.562,123.286,-61.483,177.316,15.006,151.731
C02482=1101.568,123.536,-61.502,177.319,15.007,151.731
C02483=1101.574,123.785,-61.522,177.322,15.006,151.730
C02484=1101.579,124.034,-61.541,177.326,15.006,151.729
C02485=1101.585,124.283,-61.561,177.328,15.006,151.728
C02486=1101.590,124.533,-61.581,177.332,15.006,151.728
C02487=1101.596,124.782,-61.600,177.335,15.005,151.727
C02488=1101.602,125.031,-61.620,177.338,15.005,151.726
C02489=1101.608,125.280,-61.639,177.341,15.005,151.725
C02490=1101.614,125.529,-61.659,177.345,15.005,151.725
C02491=1101.619,125.779,-61.679,177.348,15.004,151.724
C02492=1101.625,126.027,-61.698,177.351,15.004,151.723
C02493=1101.630,126.276,-61.718,177.354,15.004,151.722
C02494=1101.635,126.526,-61.737,177.357,15.004,151.722
C02495=1101.641,126.775,-61.757,177.361,15.003,151.721
C02496=1101.647,127.024,-61.776,177.364,15.003,151.720
C02497=1101.653,127.273,-61.796,177.368,15.003,151.719
C02498=1101.659,127.522,-61.816,177.371,15.002,151.719
C02499=1101.665,127.795,-61.838,177.374,15.003,151.718
C02500=1101.671,128.068,-61.860,177.378,15.002,151.717
C02501=1101.677,128.341,-61.881,177.381,15.002,151.716
C02502=1101.684,128.614,-61.903,177.385,15.001,151.715
C02503=1101.690,128.863,-61.923,177.388,15.001,151.714
C02504=1101.695,129.113,-61.943,177.391,15.001,151.714
C02505=1101.701,129.361,-61.962,177.395,15.001,151.713
C02506=1101.707,129.612,-61.982,177.398,15.000,151.712
C02507=1101.713,129.860,-62.002,177.401,15.000,151.711
C02508=1101.719,130.109,-62.022,177.404,14.999,151.711
C02509=1101.724,130.359,-62.042,177.408,15.000,151.710
C02510=1101.730,130.608,-62.062,177.411,14.999,151.709
C02511=1101.736,130.857,-62.082,177.414,14.999,151.708
C02512=1101.742,131.106,-62.101,177.417,14.998,151.707
C02513=1101.747,131.355,-62.122,177.421,14.998,151.707
C02514=1101.753,131.604,-62.142,177.424,14.998,151.706
C02515=1101.759,131.853,-62.161,177.427,14.998,151.705
C02516=1101.765,132.102,-62.181,177.431,14.997,151.704
C02517=1101.770,132.351,-62.201,177.434,14.997,151.704
C02518=1101.776,132.601,-62.221,177.437,14.996,151.703
C02519=1101.781,132.850,-62.241,177.441,14.996,151.702
C02520=1101.787,133.099,-62.261,177.444,14.995,151.701
C02521=1101.793,133.347,-62.281,177.447,14.995,151.700
C02522=1101.798,133.597,-62.301,177.450,14.995,151.700
C02523=1101.804,133.847,-62.321,177.454,14.995,151.699
C02524=1101.810,134.096,-62.342,177.456,14.995,151.698
C02525=1101.816,134.345,-62.362,177.460,14.994,151.697
C02526=1101.821,134.594,-62.382,177.463,14.994,151.697
C02527=1101.827,134.843,-62.401,177.467,14.994,151.696
C02528=1101.832,135.092,-62.422,177.470,14.993,151.695
C02529=1101.838,135.341,-62.442,177.473,14.993,151.694
C02530=1101.843,135.590,-62.463,177.477,14.993,151.693
C02531=1101.849,135.839,-62.483,177.480,14.992,151.693
C02532=1101.855,136.088,-62.502,177.484,14.992,151.692
C02533=1101.860,136.337,-62.523,177.487,14.992,151.691
C02534=1101.867,136.587,-62.543,177.490,14.992,151.690
C02535=1101.872,136.836,-62.563,177.493,14.991,151.689
C02536=1101.878,137.085,-62.583,177.497,14.991,151.689
C02537=1101.883,137.334,-62.604,177.500,14.990,151.688
C02538=1101.889,137.583,-62.624,177.504,14.990,151.687
C02539=1101.894,137.832,-62.644,177.506,14.989,151.686
C02540=1101.900,138.081,-62.664,177.510,14.989,151.685
C02541=1101.906,138.331,-62.685,177.513,14.988,151.685
C02542=1101.911,138.580,-62.706,177.517,14.988,151.684
C02543=1101.917,138.829,-62.726,177.520,14.988,151.683
C02544=1101.923,139.078,-62.746,177.523,14.988,151.682
C02545=1101.929,139.327,-62.766,177.527,14.987,151.681
C02546=1101.934,139.576,-62.787,177.530,14.987,151.681
C02547=1101.941,139.825,-62.807,177.534,14.986,151.680
C02548=1101.946,140.074,-62.828,177.537,14.986,151.679
C02549=1101.951,140.324,-62.848,177.541,14.986,151.678
C02550=1101.957,140.572,-62.868,177.544,14.985,151.677
C02551=1101.962,140.821,-62.889,177.547,14.985,151.676
C02552=1101.968,141.071,-62.909,177.550,14.984,151.676
C02553=1101.974,141.320,-62.929,177.554,14.984,151.675
C02554=1101.979,141.569,-62.950,177.557,14.983,151.674
C02555=1101.985,141.818,-62.971,177.561,14.983,151.673
C02556=1101.991,142.067,-62.991,177.564,14.982,151.672
C02557=1101.996,142.316,-63.012,177.567,14.983,151.672
C02558=1102.002,142.566,-63.033,177.570,14.982,151.671
C02559=1102.008,142.814,-63.053,177.574,14.982,151.670
C02560=1102.013,143.063,-63.073,177.578,14.981,151.669
C02561=1102.019,143.313,-63.094,177.581,14.981,151.668
C02562=1102.024,143.561,-63.115,177.585,14.981,151.667
C02563=1102.031,143.835,-63.137,177.588,14.980,151.667
C02564=1102.037,144.108,-63.160,177.592,14.979,151.666
C02565=1102.043,144.380,-63.183,177.595,14.979,151.665
C02566=1102.049,144.653,-63.205,177.599,14.979,151.664
C02567=1102.056,144.902,-63.226,177.602,14.978,151.663
C02568=1102.061,145.151,-63.247,177.606,14.978,151.662
C02569=1102.066,145.400,-63.267,177.609,14.977,151.661
C02570=1102.072,145.649,-63.288,177.613,14.977,151.661
C02571=1102.077,145.899,-63.309,177.616,14.976,151.660
C02572=1102.084,146.147,-63.329,177.620,14.976,151.659
C02573=1102.089,146.396,-63.350,177.623,14.976,151.658
C02574=1102.095,146.646,-63.371,177.627,14.975,151.657
C02575=1102.100,146.895,-63.392,177.630,14.974,151.656
C02576=1102.106,147.143,-63.412,177.633,14.974,151.655
C02577=1102.112,147.393,-63.433,177.637,14.974,151.655
C02578=1102.118,147.642,-63.454,177.640,14.973,151.654
C02579=1102.123,147.891,-63.475,177.644,14.972,151.653
C02580=1102.128,148.140,-63.495,177.647,14.972,151.652
C02581=1102.135,148.389,-63.517,177.651,14.971,151.651
C02582=1102.141,148.638,-63.537,177.654,14.970,151.650
C02583=1102.146,148.887,-63.558,177.658,14.971,151.649
C02584=1102.152,149.136,-63.579,177.661,14.970,151.649
C02585=1102.157,149.385,-63.600,177.665,14.969,151.648
C02586=1102.163,149.634,-63.621,177.669,14.969,151.647
C02587=1102.169,149.884,-63.642,177.671,14.969,151.646
C02588=1102.174,150.132,-63.663,177.675,14.968,151.645
C02589=1102.179,150.381,-63.684,177.678,14.967,151.644
C02590=1102.186,150.631,-63.705,177.682,14.967,151.644
C02591=1102.191,150.880,-63.726,177.685,14.966,151.643
C02592=1102.196,151.128,-63.747,177.689,14.966,151.642
C02593=1102.202,151.378,-63.768,177.692,14.965,151.641
C02594=1102.208,151.627,-63.789,177.696,14.965,151.640
C02595=1102.214,151.876,-63.810,177.700,14.965,151.639
C02596=1102.219,152.125,-63.832,177.703,14.964,151.638
C02597=1102.224,152.374,-63.852,177.707,14.964,151.637
C02598=1102.231,152.623,-63.874,177.710,14.963,151.636
C02599=1102.236,152.872,-63.894,177.714,14.962,151.636
C02600=1102.241,153.121,-63.916,177.716,14.962,151.635
C02601=1102.248,153.370,-63.937,177.720,14.962,151.634
C02602=1102.253,153.619,-63.958,177.723,14.961,151.633
C02603=1102.259,153.868,-63.980,177.727,14.960,151.632
C02604=1102.264,154.118,-64.000,177.731,14.960,151.631
C02605=1102.270,154.366,-64.021,177.734,14.959,151.630
C02606=1102.276,154.615,-64.043,177.738,14.959,151.629
C02607=1102.281,154.864,-64.064,177.741,14.958,151.629
C02608=1102.287,155.114,-64.085,177.745,14.957,151.628
C02609=1102.293,155.362,-64.106,177.748,14.957,151.627
C02610=1102.299,155.611,-64.128,177.752,14.957,151.626
C02611=1102.304,155.860,-64.149,177.755,14.956,151.625
C02612=1102.311,156.110,-64.170,177.759,14.955,151.624
C02613=1102.316,156.358,-64.192,177.763,14.955,151.623
C02614=1102.321,156.608,-64.213,177.766,14.954,151.622
C02615=1102.327,156.857,-64.234,177.770,14.954,151.621
C02616=1102.332,157.105,-64.256,177.773,14.953,151.621
C02617=1102.339,157.354,-64.277,177.777,14.953,151.620
C02618=1102.344,157.604,-64.298,177.780,14.952,151.619
C02619=1102.350,157.853,-64.319,177.784,14.951,151.618
C02620=1102.355,158.102,-64.341,177.788,14.951,151.617
C02621=1102.361,158.351,-64.363,177.791,14.950,151.616
C02622=1102.367,158.599,-64.384,177.795,14.950,151.615
C02623=1102.372,158.849,-64.405,177.798,14.949,151.614
C02624=1102.378,159.098,-64.426,177.802,14.949,151.613
C02625=1102.383,159.347,-64.449,177.805,14.948,151.612
C02626=1102.389,159.596,-64.470,177.809,14.947,151.612
C02627=1102.396,159.868,-64.494,177.813,14.947,151.610
C02628=1102.401,160.141,-64.517,177.817,14.946,151.610
C02629=1102.408,160.413,-64.540,177.821,14.945,151.609
C02630=1102.414,160.686,-64.564,177.824,14.945,151.608
C02631=1102.420,160.935,-64.586,177.828,14.944,151.607
C02632=1102.426,161.184,-64.607,177.831,14.943,151.606
C02633=1102.431,161.433,-64.629,177.836,14.943,151.605
C02634=1102.437,161.682,-64.651,177.839,14.942,151.604
C02635=1102.442,161.931,-64.672,177.843,14.941,151.603
C02636=1102.448,162.180,-64.694,177.847,14.941,151.602
C02637=1102.453,162.429,-64.716,177.850,14.940,151.601
C02638=1102.459,162.678,-64.736,177.854,14.940,151.600
C02639=1102.464,162.927,-64.758,177.857,14.939,151.599
C02640=1102.470,163.176,-64.780,177.861,14.939,151.598
C02641=1102.475,163.425,-64.803,177.864,14.938,151.598
C02642=1102.481,163.674,-64.824,177.868,14.937,151.597
C02643=1102.486,163.923,-64.846,177.872,14.937,151.596
C02644=1102.492,164.172,-64.868,177.875,14.936,151.595
C02645=1102.497,164.421,-64.890,177.879,14.936,151.594
C02646=1102.503,164.670,-64.911,177.882,14.935,151.593
C02647=1102.509,164.919,-64.933,177.886,14.935,151.592
C02648=1102.514,165.168,-64.955,177.890,14.934,151.591
C02649=1102.520,165.417,-64.977,177.893,14.933,151.590
C02650=1102.525,165.666,-64.998,177.897,14.933,151.589
C02651=1102.531,165.915,-65.020,177.900,14.932,151.588
C02652=1102.536,166.164,-65.042,177.904,14.932,151.587
C02653=1102.542,166.413,-65.065,177.907,14.931,151.587
C02654=1102.548,166.662,-65.086,177.911,14.930,151.586
C02655=1102.553,166.911,-65.108,177.915,14.930,151.585
C02656=1102.559,167.160,-65.130,177.918,14.929,151.584
C02657=1102.564,167.409,-65.152,177.922,14.928,151.583
C02658=1102.570,167.658,-65.173,177.925,14.928,151.582
C02659=1102.576,167.907,-65.196,177.930,14.927,151.581
C02660=1102.582,168.155,-65.217,177.933,14.927,151.580
C02661=1102.587,168.405,-65.240,177.937,14.926,151.579
C02662=1102.592,168.654,-65.262,177.940,14.925,151.578
C02663=1102.598,168.902,-65.284,177.944,14.924,151.577
C02664=1102.604,169.152,-65.306,177.948,14.924,151.576
C02665=1102.609,169.400,-65.327,177.951,14.923,151.575
C02666=1102.615,169.649,-65.350,177.955,14.922,151.574
C02667=1102.621,169.899,-65.372,177.959,14.922,151.573
C02668=1102.626,170.147,-65.394,177.962,14.921,151.572
C02669=1102.632,170.396,-65.417,177.966,14.921,151.572
C02670=1102.638,170.645,-65.438,177.969,14.919,151.570
C02671=1102.643,170.894,-65.460,177.973,14.919,151.570
C02672=1102.649,171.143,-65.483,177.977,14.919,151.569
C02673=1102.655,171.392,-65.505,177.981,14.917,151.568
C02674=1102.659,171.641,-65.527,177.985,14.917,151.567
C02675=1102.666,171.890,-65.549,177.988,14.916,151.566
C02676=1102.671,172.139,-65.571,177.992,14.915,151.565
C02677=1102.677,172.388,-65.594,177.995,14.915,151.564
C02678=1102.683,172.637,-65.616,177.999,14.914,151.563
C02679=1102.688,172.886,-65.638,178.003,14.914,151.562
C02680=1102.694,173.135,-65.661,178.007,14.912,151.561
C02681=1102.700,173.384,-65.682,178.011,14.912,151.560
C02682=1102.705,173.632,-65.705,178.014,14.911,151.559
C02683=1102.710,173.882,-65.727,178.018,14.910,151.558
C02684=1102.717,174.131,-65.750,178.022,14.910,151.557
C02685=1102.722,174.380,-65.772,178.025,14.909,151.556
C02686=1102.728,174.628,-65.794,178.029,14.908,151.555
C02687=1102.734,174.878,-65.816,178.033,14.907,151.554
C02688=1102.739,175.126,-65.839,178.036,14.907,151.553
C02689=1102.745,175.375,-65.862,178.041,14.906,151.552
C02690=1102.751,175.624,-65.883,178.044,14.905,151.551
C02691=1102.757,175.896,-65.908,178.048,14.905,151.550
C02692=1102.763,176.168,-65.932,178.052,14.904,151.549
C02693=1102.770,176.441,-65.957,178.057,14.903,151.548
C02694=1102.776,176.713,-65.982,178.060,14.901,151.547
C02695=1102.781,176.962,-66.004,178.064,14.901,151.546
C02696=1102.787,177.211,-66.027,178.068,14.900,151.545
C02697=1102.793,177.460,-66.049,178.071,14.899,151.544
C02698=1102.799,177.709,-66.071,178.076,14.899,151.543
C02699=1102.804,177.958,-66.094,178.079,14.897,151.542
C02700=1102.810,178.207,-66.117,178.083,14.897,151.541
C02701=1102.815,178.456,-66.139,178.087,14.896,151.540
C02702=1102.821,178.704,-66.162,178.090,14.896,151.539
C02703=1102.827,178.953,-66.185,178.095,14.895,151.538
C02704=1102.833,179.202,-66.207,178.098,14.894,151.537
C02705=1102.838,179.452,-66.230,178.102,14.893,151.536
C02706=1102.845,179.700,-66.252,178.105,14.892,151.535
C02707=1102.850,179.949,-66.275,178.110,14.891,151.534
C02708=1102.856,180.198,-66.298,178.113,14.891,151.533
C02709=1102.862,180.447,-66.320,178.117,14.890,151.532
C02710=1102.867,180.696,-66.343,178.121,14.889,151.531
C02711=1102.873,180.945,-66.366,178.125,14.888,151.530
C02712=1102.879,181.193,-66.388,178.128,14.887,151.529
C02713=1102.885,181.442,-66.411,178.133,14.887,151.528
C02714=1102.890,181.691,-66.434,178.136,14.885,151.527
C02715=1102.896,181.940,-66.456,178.140,14.885,151.526
C02716=1102.902,182.189,-66.479,178.144,14.884,151.525
C02717=1102.907,182.438,-66.502,178.148,14.883,151.524
C02718=1102.914,182.687,-66.524,178.152,14.882,151.523
C02719=1102.920,182.936,-66.547,178.155,14.881,151.522
C02720=1102.925,183.185,-66.570,178.159,14.881,151.521
C02721=1102.931,183.434,-66.593,178.163,14.880,151.520
C02722=1102.937,183.682,-66.616,178.167,14.879,151.519
C02723=1102.942,183.931,-66.639,178.171,14.878,151.517
C02724=1102.948,184.180,-66.662,178.175,14.877,151.516
C02725=1102.954,184.429,-66.685,178.179,14.876,151.515
C02726=1102.960,184.678,-66.708,178.182,14.875,151.514
C02727=1102.966,184.927,-66.730,178.186,14.875,151.513
C02728=1102.972,185.176,-66.753,178.190,14.874,151.512
C02729=1102.977,185.425,-66.777,178.194,14.873,151.511
C02730=1102.983,185.674,-66.800,178.198,14.872,151.510
C02731=1102.988,185.923,-66.823,178.201,14.871,151.509
C02732=1102.994,186.171,-66.846,178.205,14.870,151.508
C02733=1103.000,186.420,-66.869,178.210,14.870,151.507
C02734=1103.005,186.669,-66.892,178.213,14.869,151.506
C02735=1103.010,186.918,-66.915,178.217,14.868,151.505
C02736=1103.016,187.167,-66.938,178.220,14.867,151.504
C02737=1103.021,187.415,-66.961,178.225,14.866,151.503
C02738=1103.027,187.664,-66.984,178.228,14.866,151.502
C02739=1103.033,187.913,-67.007,178.232,14.865,151.501
C02740=1103.038,188.162,-67.031,178.236,14.864,151.500
C02741=1103.044,188.411,-67.054,178.240,14.863,151.499
C02742=1103.050,188.660,-67.077,178.244,14.862,151.498
C02743=1103.055,188.909,-67.100,178.248,14.862,151.497
C02744=1103.061,189.157,-67.123,178.251,14.860,151.496
C02745=1103.066,189.407,-67.146,178.255,14.860,151.495
C02746=1103.072,189.655,-67.170,178.260,14.859,151.494
C02747=1103.078,189.904,-67.193,178.263,14.858,151.493
C02748=1103.084,190.153,-67.216,178.267,14.857,151.492
C02749=1103.089,190.402,-67.239,178.270,14.856,151.491
C02750=1103.094,190.651,-67.262,178.275,14.856,151.490
C02751=1103.100,190.899,-67.286,178.279,14.855,151.489
C02752=1103.105,191.148,-67.309,178.282,14.854,151.488
C02753=1103.111,191.397,-67.332,178.286,14.853,151.487
C02754=1103.117,191.645,-67.356,178.291,14.852,151.486
C02755=1103.123,191.918,-67.382,178.294,14.851,151.485
C02756=1103.130,192.190,-67.407,178.299,14.850,151.483
C02757=1103.135,192.462,-67.432,178.303,14.849,151.482
C02758=1103.142,192.734,-67.458,178.307,14.848,151.481
C02759=1103.148,192.983,-67.481,178.312,14.848,151.480
C02760=1103.153,193.231,-67.505,178.315,14.846,151.479
C02761=1103.159,193.480,-67.528,178.319,14.846,151.478
C02762=1103.164,193.729,-67.551,178.323,14.844,151.477
C02763=1103.170,193.978,-67.576,178.327,14.844,151.476
C02764=1103.176,194.226,-67.599,178.331,14.843,151.475
C02765=1103.182,194.475,-67.622,178.335,14.842,151.474
C02766=1103.187,194.725,-67.646,178.339,14.841,151.473
C02767=1103.193,194.974,-67.669,178.343,14.840,151.471
C02768=1103.199,195.222,-67.693,178.347,14.839,151.470
C02769=1103.204,195.471,-67.716,178.351,14.838,151.469
C02770=1103.210,195.719,-67.740,178.354,14.837,151.468
C02771=1103.215,195.969,-67.763,178.358,14.837,151.467
C02772=1103.221,196.217,-67.787,178.363,14.836,151.466
C02773=1103.227,196.466,-67.810,178.366,14.835,151.465
C02774=1103.233,196.715,-67.835,178.370,14.834,151.464
C02775=1103.239,196.963,-67.858,178.374,14.833,151.463
C02776=1103.244,197.212,-67.882,178.378,14.832,151.462
C02777=1103.250,197.461,-67.906,178.382,14.831,151.461
C02778=1103.256,197.710,-67.929,178.386,14.830,151.460
C02779=1103.261,197.959,-67.953,178.390,14.829,151.459
C02780=1103.267,198.208,-67.976,178.394,14.828,151.458
C02781=1103.272,198.456,-68.000,178.398,14.827,151.457
C02782=1103.278,198.705,-68.024,178.402,14.826,151.455
C02783=1103.284,198.955,-68.048,178.406,14.826,151.454
C02784=1103.290,199.203,-68.072,178.410,14.825,151.453
C02785=1103.296,199.451,-68.095,178.414,14.823,151.452
C02786=1103.301,199.700,-68.119,178.418,14.822,151.451
C02787=1103.308,199.949,-68.143,178.422,14.822,151.450
C02788=1103.313,200.198,-68.167,178.426,14.821,151.449
C02789=1103.319,200.447,-68.190,178.430,14.820,151.448
C02790=1103.324,200.695,-68.214,178.434,14.819,151.447
C02791=1103.331,200.944,-68.238,178.438,14.818,151.446
C02792=1103.336,201.193,-68.262,178.442,14.817,151.445
C02793=1103.342,201.442,-68.285,178.446,14.816,151.444
C02794=1103.348,201.691,-68.310,178.450,14.814,151.442
C02795=1103.354,201.939,-68.334,178.454,14.814,151.441
C02796=1103.359,202.188,-68.358,178.458,14.813,151.440
C02797=1103.366,202.437,-68.382,178.462,14.812,151.439
C02798=1103.371,202.686,-68.406,178.466,14.811,151.438
C02799=1103.376,202.935,-68.430,178.470,14.810,151.437
C02800=1103.382,203.183,-68.453,178.474,14.809,151.436
C02801=1103.388,203.432,-68.478,178.478,14.808,151.435
C02802=1103.393,203.681,-68.502,178.482,14.808,151.434
C02803=1103.399,203.929,-68.526,178.486,14.806,151.432
C02804=1103.405,204.179,-68.550,178.490,14.805,151.431
C02805=1103.410,204.428,-68.574,178.494,14.804,151.430
C02806=1103.416,204.676,-68.598,178.498,14.803,151.429
C02807=1103.421,204.925,-68.622,178.502,14.802,151.428
C02808=1103.427,205.174,-68.647,178.506,14.801,151.427
C02809=1103.433,205.422,-68.671,178.510,14.800,151.426
C02810=1103.439,205.671,-68.695,178.514,14.800,151.425
C02811=1103.444,205.920,-68.719,178.518,14.798,151.424
C02812=1103.450,206.169,-68.743,178.522,14.798,151.423
C02813=1103.455,206.417,-68.768,178.526,14.797,151.422
C02814=1103.462,206.666,-68.792,178.530,14.796,151.421
C02815=1103.467,206.915,-68.816,178.534,14.795,151.419
C02816=1103.473,207.164,-68.841,178.538,14.793,151.418
C02817=1103.478,207.413,-68.865,178.542,14.793,151.417
C02818=1103.484,207.661,-68.889,178.547,14.792,151.416
C02819=1103.508,208.661,-68.987,178.576,14.795,151.410
C02820=1103.515,209.029,-69.023,178.583,14.795,151.409
C02821=1103.524,209.396,-69.059,178.588,14.795,151.408
C02822=1103.532,209.764,-69.095,178.593,14.795,151.406
C02823=1103.540,210.131,-69.132,178.599,14.795,151.405
C02824=1103.546,210.380,-69.156,178.602,14.794,151.404
C02825=1103.552,210.629,-69.181,178.606,14.794,151.403
C02826=1103.557,210.877,-69.205,178.610,14.794,151.402
C02827=1103.563,211.125,-69.229,178.614,14.793,151.402
C02828=1103.569,211.375,-69.254,178.618,14.794,151.401
C02829=1103.575,211.623,-69.279,178.621,14.794,151.400
C02830=1103.581,211.872,-69.303,178.625,14.793,151.399
C02831=1103.585,212.121,-69.328,178.629,14.793,151.398
C02832=1103.591,212.369,-69.353,178.633,14.793,151.397
C02833=1103.597,212.618,-69.378,178.637,14.793,151.396
C02834=1103.603,212.867,-69.402,178.641,14.793,151.396
C02835=1103.608,213.115,-69.427,178.644,14.793,151.395
C02836=1103.614,213.365,-69.452,178.648,14.793,151.394
C02837=1103.619,213.613,-69.476,178.652,14.793,151.393
C02838=1103.626,213.862,-69.502,178.656,14.792,151.392
C02839=1103.631,214.110,-69.526,178.660,14.793,151.391
C02840=1103.637,214.359,-69.551,178.663,14.793,151.391
C02841=1103.642,214.608,-69.575,178.667,14.792,151.390
C02842=1103.648,214.857,-69.600,178.670,14.792,151.389
C02843=1103.653,215.105,-69.626,178.674,14.791,151.388
C02844=1103.659,215.355,-69.650,178.678,14.792,151.387
C02845=1103.665,215.603,-69.675,178.682,14.792,151.386
C02846=1103.671,215.852,-69.700,178.686,14.791,151.385
C02847=1103.676,216.100,-69.725,178.690,14.791,151.385
C02848=1103.682,216.349,-69.749,178.693,14.791,151.384
C02849=1103.687,216.597,-69.775,178.697,14.791,151.383
C02850=1103.693,216.847,-69.800,178.701,14.791,151.382
C02851=1103.698,217.095,-69.825,178.705,14.791,151.381
C02852=1103.704,217.344,-69.849,178.709,14.791,151.380
C02853=1103.709,217.592,-69.875,178.713,14.791,151.379
C02854=1103.715,217.841,-69.900,178.716,14.791,151.379
C02855=1103.721,218.090,-69.925,178.720,14.791,151.378
C02856=1103.727,218.338,-69.950,178.724,14.791,151.377
C02857=1103.733,218.587,-69.974,178.728,14.791,151.376
C02858=1103.738,218.836,-70.000,178.732,14.790,151.375
C02859=1103.744,219.084,-70.025,178.735,14.791,151.374
C02860=1103.750,219.334,-70.050,178.739,14.791,151.374
C02861=1103.755,219.582,-70.075,178.743,14.790,151.373
C02862=1103.761,219.831,-70.101,178.747,14.790,151.372
C02863=1103.766,220.079,-70.125,178.751,14.790,151.371
C02864=1103.772,220.328,-70.150,178.754,14.790,151.370
C02865=1103.778,220.577,-70.176,178.758,14.790,151.369
C02866=1103.783,220.825,-70.201,178.762,14.790,151.368
C02867=1103.789,221.074,-70.226,178.766,14.790,151.367
C02868=1103.796,221.323,-70.251,178.770,14.790,151.367
C02869=1103.800,221.571,-70.277,178.774,14.790,151.366
C02870=1103.807,221.820,-70.302,178.777,14.790,151.365
C02871=1103.813,222.069,-70.327,178.781,14.790,151.364
C02872=1103.821,222.440,-70.365,178.786,14.789,151.363
C02873=1103.829,222.811,-70.403,178.792,14.790,151.362
C02874=1103.837,223.181,-70.441,178.798,14.789,151.360
C02875=1103.846,223.552,-70.478,178.804,14.790,151.359
C02876=1103.851,223.801,-70.504,178.807,14.790,151.358
C02877=1103.857,224.050,-70.530,178.811,14.789,151.357
C02878=1103.863,224.298,-70.555,178.815,14.789,151.357
C02879=1103.868,224.547,-70.580,178.819,14.790,151.356
C02880=1103.874,224.796,-70.605,178.823,14.789,151.355
C02881=1103.879,225.044,-70.631,178.827,14.789,151.354
C02882=1103.885,225.293,-70.656,178.830,14.789,151.353
C02883=1103.891,225.542,-70.682,178.834,14.789,151.352
C02884=1103.897,225.791,-70.707,178.838,14.789,151.352
C02885=1103.902,226.039,-70.733,178.842,14.789,151.351
C02886=1103.907,226.288,-70.759,178.846,14.789,151.350
C02887=1103.914,226.537,-70.784,178.849,14.789,151.349
C02888=1103.919,226.786,-70.810,178.853,14.789,151.348
C02889=1103.925,227.033,-70.835,178.857,14.789,151.347
C02890=1103.930,227.282,-70.861,178.861,14.789,151.346
C02891=1103.936,227.531,-70.886,178.864,14.789,151.346
C02892=1103.942,227.780,-70.912,178.868,14.789,151.345
C02893=1103.947,228.028,-70.937,178.872,14.789,151.344
C02894=1103.953,228.276,-70.964,178.876,14.789,151.343
C02895=1103.959,228.525,-70.990,178.879,14.789,151.342
C02896=1103.965,228.774,-71.015,178.883,14.789,151.341
C02897=1103.970,229.023,-71.041,178.887,14.789,151.341
C02898=1103.976,229.271,-71.066,178.891,14.789,151.340
C02899=1103.981,229.520,-71.092,178.895,14.789,151.339
C02900=1103.988,229.769,-71.117,178.898,14.789,151.338
C02901=1103.993,230.017,-71.144,178.902,14.789,151.337
C02902=1103.999,230.266,-71.170,178.906,14.789,151.336
C02903=1104.004,230.514,-71.195,178.910,14.789,151.336
C02904=1104.010,230.763,-71.221,178.914,14.789,151.335
C02905=1104.015,231.012,-71.247,178.918,14.789,151.334
C02906=1104.021,231.260,-71.273,178.921,14.789,151.333
C02907=1104.027,231.509,-71.299,178.925,14.789,151.332
C02908=1104.033,231.758,-71.325,178.929,14.789,151.331
C02909=1104.038,232.006,-71.350,178.933,14.790,151.331
C02910=1104.044,232.254,-71.376,178.937,14.790,151.330
C02911=1104.050,232.503,-71.402,178.941,14.789,151.329
C02912=1104.055,232.752,-71.428,178.944,14.790,151.328
C02913=1104.061,233.001,-71.455,178.948,14.790,151.327
C02914=1104.066,233.250,-71.481,178.952,14.789,151.326
C02915=1104.073,233.498,-71.506,178.956,14.790,151.326
C02916=1104.078,233.746,-71.532,178.960,14.790,151.325
C02917=1104.083,233.995,-71.558,178.963,14.790,151.324
C02918=1104.089,234.243,-71.585,178.967,14.790,151.323
C02919=1104.094,234.492,-71.611,178.971,14.790,151.322
C02920=1104.100,234.741,-71.637,178.975,14.790,151.322
C02921=1104.106,234.989,-71.663,178.978,14.790,151.321
C02922=1104.112,235.238,-71.689,178.982,14.790,151.320
C02923=1104.118,235.487,-71.715,178.986,14.790,151.319
C02924=1104.126,235.849,-71.753,178.992,14.790,151.318
C02925=1104.133,236.211,-71.791,178.997,14.790,151.317
C02926=1104.142,236.574,-71.829,179.003,14.791,151.316
C02927=1104.149,236.937,-71.868,179.008,14.791,151.315
C02928=1104.155,237.185,-71.894,179.013,14.791,151.314
C02929=1104.161,237.434,-71.920,179.016,14.791,151.313
C02930=1104.167,237.682,-71.946,179.020,14.791,151.312
C02931=1104.173,237.931,-71.972,179.024,14.791,151.311
C02932=1104.178,238.179,-71.999,179.028,14.791,151.310
C02933=1104.184,238.428,-72.026,179.031,14.792,151.310
C02934=1104.190,238.677,-72.052,179.035,14.791,151.309
C02935=1104.195,238.925,-72.078,179.039,14.792,151.308
C02936=1104.201,239.173,-72.105,179.042,14.792,151.307
C02937=1104.207,239.422,-72.131,179.046,14.792,151.306
C02938=1104.212,239.671,-72.158,179.050,14.792,151.306
C02939=1104.218,239.919,-72.184,179.055,14.792,151.305
C02940=1104.224,240.168,-72.210,179.058,14.792,151.304
C02941=1104.230,240.416,-72.237,179.062,14.793,151.303
C02942=1104.235,240.665,-72.263,179.066,14.793,151.302
C02943=1104.241,240.914,-72.289,179.069,14.793,151.302
C02944=1104.247,241.162,-72.316,179.073,14.793,151.301
C02945=1104.252,241.410,-72.343,179.077,14.793,151.300
C02946=1104.258,241.659,-72.369,179.081,14.793,151.299
C02947=1104.264,241.907,-72.396,179.084,14.793,151.298
C02948=1104.269,242.156,-72.422,179.089,14.794,151.297
C02949=1104.274,242.405,-72.449,179.093,14.794,151.297
C02950=1104.280,242.653,-72.476,179.097,14.794,151.296
C02951=1104.286,242.902,-72.502,179.100,14.794,151.295
C02952=1104.292,243.151,-72.529,179.104,14.794,151.294
C02953=1104.298,243.400,-72.555,179.107,14.794,151.293
C02954=1104.304,243.648,-72.582,179.111,14.794,151.293
C02955=1104.309,243.896,-72.609,179.115,14.794,151.292
C02956=1104.314,244.145,-72.636,179.119,14.795,151.291
C02957=1104.320,244.393,-72.663,179.123,14.795,151.290
C02958=1104.326,244.642,-72.689,179.127,14.795,151.289
C02959=1104.332,244.890,-72.716,179.130,14.796,151.289
C02960=1104.337,245.138,-72.742,179.134,14.795,151.288
C02961=1104.342,245.387,-72.770,179.138,14.796,151.287
C02962=1104.348,245.635,-72.796,179.142,14.796,151.286
C02963=1104.354,245.884,-72.823,179.146,14.796,151.285
C02964=1104.360,246.132,-72.850,179.150,14.797,151.285
C02965=1104.365,246.381,-72.877,179.154,14.796,151.284
C02966=1104.371,246.630,-72.904,179.157,14.797,151.283
C02967=1104.377,246.878,-72.931,179.161,14.797,151.282
C02968=1104.382,247.127,-72.958,179.165,14.797,151.282
C02969=1104.388,247.375,-72.984,179.169,14.797,151.281
C02970=1104.394,247.624,-73.011,179.173,14.798,151.280
C02971=1104.399,247.872,-73.038,179.176,14.798,151.279
C02972=1104.404,248.121,-73.065,179.180,14.798,151.278
C02973=1104.410,248.369,-73.092,179.184,14.798,151.278
C02974=1104.415,248.618,-73.119,179.188,14.798,151.277
C02975=1104.422,248.867,-73.146,179.191,14.799,151.276
C02976=1104.429,249.223,-73.185,179.197,14.800,151.275
C02977=1104.437,249.578,-73.223,179.202,14.799,151.274
C02978=1104.445,249.934,-73.262,179.208,14.800,151.273
C02979=1104.454,250.290,-73.301,179.213,14.801,151.272
C02980=1104.459,250.538,-73.329,179.217,14.801,151.271
C02981=1104.465,250.786,-73.356,179.221,14.801,151.270
C02982=1104.470,251.035,-73.383,179.224,14.802,151.269
C02983=1104.476,251.283,-73.410,179.228,14.801,151.269
C02984=1104.481,251.531,-73.438,179.232,14.802,151.268
C02985=1104.487,251.780,-73.465,179.236,14.802,151.267
C02986=1104.492,252.029,-73.492,179.240,14.803,151.266
C02987=1104.498,252.277,-73.519,179.243,14.803,151.266
C02988=1104.503,252.526,-73.546,179.247,14.803,151.265
C02989=1104.509,252.774,-73.573,179.251,14.803,151.264
C02990=1104.515,253.023,-73.601,179.255,14.804,151.263
C02991=1104.521,253.271,-73.628,179.259,14.804,151.262
C02992=1104.526,253.520,-73.655,179.263,14.805,151.262
C02993=1104.532,253.767,-73.683,179.266,14.805,151.261
C02994=1104.538,254.017,-73.710,179.270,14.805,151.260
C02995=1104.543,254.265,-73.737,179.273,14.805,151.260
C02996=1104.549,254.513,-73.765,179.278,14.806,151.259
C02997=1104.555,254.762,-73.792,179.282,14.806,151.258
C02998=1104.560,255.010,-73.820,179.285,14.806,151.257
C02999=1104.565,255.259,-73.847,179.289,14.806,151.256
C03000=1104.572,255.507,-73.875,179.293,14.807,151.256
C03001=1104.577,255.755,-73.902,179.297,14.807,151.255
C03002=1104.583,256.004,-73.929,179.301,14.808,151.254
C03003=1104.588,256.252,-73.957,179.304,14.808,151.253
C03004=1104.594,256.501,-73.985,179.308,14.808,151.253
C03005=1104.600,256.750,-74.012,179.312,14.809,151.252
C03006=1104.605,256.998,-74.040,179.316,14.809,151.251
C03007=1104.611,257.246,-74.066,179.320,14.809,151.250
C03008=1104.617,257.495,-74.095,179.323,14.810,151.250
C03009=1104.622,257.743,-74.123,179.327,14.810,151.249
C03010=1104.628,257.991,-74.149,179.331,14.811,151.248
C03011=1104.634,258.240,-74.178,179.335,14.811,151.247
C03012=1104.639,258.488,-74.206,179.339,14.811,151.246
C03013=1104.645,258.736,-74.232,179.342,14.811,151.246
C03014=1104.651,258.985,-74.260,179.346,14.812,151.245
C03015=1104.657,259.233,-74.288,179.350,14.812,151.244
C03016=1104.663,259.482,-74.315,179.354,14.813,151.243
C03017=1104.668,259.730,-74.343,179.358,14.812,151.243
C03018=1104.674,259.978,-74.371,179.361,14.813,151.242
C03019=1104.680,260.227,-74.398,179.366,14.814,151.241
C03020=1104.685,260.475,-74.426,179.370,14.814,151.240
C03021=1104.691,260.724,-74.455,179.373,14.814,151.240
C03022=1104.697,260.972,-74.482,179.377,14.814,151.239
C03023=1104.703,261.220,-74.510,179.380,14.814,151.238
C03024=1104.708,261.469,-74.538,179.385,14.815,151.237
C03025=1104.714,261.717,-74.566,179.388,14.816,151.237
C03026=1104.720,261.966,-74.593,179.392,14.816,151.236
C03027=1104.726,262.214,-74.621,179.396,14.816,151.235
C03028=1104.734,262.567,-74.661,179.401,14.817,151.234
C03029=1104.743,262.920,-74.701,179.407,14.818,151.233
C03030=1104.750,263.273,-74.740,179.412,14.818,151.232
C03031=1104.759,263.626,-74.780,179.418,14.819,151.231
C03032=1104.764,263.875,-74.808,179.421,14.819,151.230
C03033=1104.770,264.123,-74.836,179.425,14.819,151.229
C03034=1104.776,264.372,-74.864,179.430,14.820,151.229
C03035=1104.782,264.620,-74.892,179.433,14.820,151.228
C03036=1104.787,264.868,-74.920,179.437,14.821,151.227
C03037=1104.793,265.116,-74.948,179.440,14.821,151.227
C03038=1104.798,265.365,-74.976,179.444,14.822,151.226
C03039=1104.804,265.613,-75.004,179.448,14.822,151.225
C03040=1104.810,265.861,-75.032,179.452,14.822,151.224
C03041=1104.816,266.110,-75.060,179.455,14.823,151.224
C03042=1104.821,266.357,-75.089,179.460,14.824,151.223
C03043=1104.827,266.606,-75.117,179.463,14.824,151.222
C03044=1104.832,266.854,-75.145,179.467,14.824,151.221
C03045=1104.838,267.103,-75.174,179.470,14.825,151.221
C03046=1104.844,267.351,-75.202,179.474,14.826,151.220
C03047=1104.850,267.600,-75.230,179.478,14.826,151.219
C03048=1104.855,267.848,-75.258,179.482,14.826,151.219
C03049=1104.861,268.097,-75.286,179.486,14.827,151.218
C03050=1104.866,268.345,-75.314,179.490,14.828,151.217
C03051=1104.873,268.593,-75.343,179.493,14.828,151.216
C03052=1104.878,268.841,-75.371,179.497,14.828,151.216
C03053=1104.883,269.090,-75.400,179.501,14.829,151.215
C03054=1104.888,269.338,-75.428,179.505,14.829,151.214
C03055=1104.894,269.587,-75.456,179.508,14.830,151.214
C03056=1104.901,269.835,-75.485,179.513,14.831,151.213
C03057=1104.906,270.083,-75.513,179.516,14.831,151.212
C03058=1104.912,270.332,-75.542,179.520,14.831,151.211
C03059=1104.918,270.579,-75.570,179.523,14.832,151.211
C03060=1104.924,270.828,-75.599,179.527,14.833,151.210
C03061=1104.929,271.076,-75.627,179.531,14.833,151.209
C03062=1104.934,271.325,-75.656,179.535,14.834,151.209
C03063=1104.940,271.573,-75.685,179.539,14.835,151.208
C03064=1104.946,271.821,-75.713,179.542,14.835,151.207
C03065=1104.952,272.069,-75.742,179.546,14.835,151.207
C03066=1104.957,272.317,-75.770,179.550,14.836,151.206
C03067=1104.962,272.566,-75.799,179.554,14.837,151.205
C03068=1104.969,272.815,-75.828,179.557,14.837,151.205
C03069=1104.974,273.063,-75.856,179.561,14.838,151.204
C03070=1104.980,273.311,-75.885,179.565,14.838,151.203
C03071=1104.986,273.559,-75.913,179.569,14.839,151.202
C03072=1104.991,273.808,-75.941,179.573,14.840,151.202
C03073=1104.997,274.056,-75.970,179.577,14.840,151.201
C03074=1105.002,274.304,-75.998,179.580,14.840,151.200
C03075=1105.009,274.552,-76.027,179.584,14.842,151.200
C03076=1105.014,274.801,-76.056,179.588,14.842,151.199
C03077=1105.020,275.049,-76.085,179.591,14.843,151.198
C03078=1105.026,275.297,-76.113,179.595,14.844,151.198
C03079=1105.030,275.545,-76.143,179.599,14.844,151.197
C03080=1105.039,275.901,-76.184,179.605,14.845,151.196
C03081=1105.047,276.257,-76.226,179.609,14.845,151.195
C03082=1105.055,276.613,-76.267,179.615,14.846,151.194
C03083=1105.064,276.969,-76.308,179.620,14.847,151.193
C03084=1105.069,277.217,-76.337,179.624,14.848,151.192
C03085=1105.075,277.465,-76.365,179.628,14.849,151.192
C03086=1105.080,277.714,-76.395,179.632,14.849,151.191
C03087=1105.086,277.961,-76.424,179.635,14.850,151.191
C03088=1105.092,278.209,-76.453,179.639,14.851,151.190
C03089=1105.097,278.458,-76.482,179.643,14.851,151.189
C03090=1105.103,278.706,-76.510,179.646,14.852,151.188
C03091=1105.109,278.954,-76.540,179.651,14.853,151.188
C03092=1105.114,279.203,-76.568,179.654,14.853,151.187
C03093=1105.120,279.452,-76.598,179.658,14.854,151.186
C03094=1105.126,279.699,-76.627,179.662,14.855,151.186
C03095=1105.131,279.947,-76.656,179.665,14.856,151.185
C03096=1105.137,280.196,-76.685,179.669,14.857,151.185
C03097=1105.143,280.445,-76.714,179.673,14.857,151.184
C03098=1105.148,280.692,-76.743,179.676,14.857,151.183
C03099=1105.154,280.940,-76.772,179.681,14.858,151.182
C03100=1105.160,281.189,-76.802,179.684,14.859,151.182
C03101=1105.166,281.437,-76.831,179.687,14.860,151.181
C03102=1105.171,281.684,-76.860,179.692,14.861,151.181
C03103=1105.177,281.933,-76.889,179.695,14.861,151.180
C03104=1105.183,282.182,-76.918,179.699,14.862,151.179
C03105=1105.188,282.430,-76.947,179.703,14.863,151.179
C03106=1105.193,282.678,-76.977,179.706,14.863,151.178
C03107=1105.199,282.926,-77.006,179.710,14.864,151.177
C03108=1105.205,283.174,-77.035,179.714,14.865,151.177
C03109=1105.210,283.423,-77.065,179.718,14.866,151.176
C03110=1105.217,283.671,-77.094,179.721,14.867,151.175
C03111=1105.221,283.919,-77.123,179.725,14.867,151.175
C03112=1105.228,284.167,-77.152,179.729,14.869,151.174
C03113=1105.233,284.415,-77.182,179.732,14.869,151.174
C03114=1105.239,284.664,-77.212,179.737,14.870,151.173
C03115=1105.245,284.912,-77.241,179.740,14.871,151.172
C03116=1105.250,285.160,-77.270,179.743,14.871,151.172
C03117=1105.255,285.408,-77.300,179.748,14.872,151.171
C03118=1105.261,285.656,-77.330,179.751,14.873,151.171
C03119=1105.268,285.904,-77.359,179.755,14.874,151.170
C03120=1105.273,286.152,-77.389,179.759,14.875,151.169
C03121=1105.279,286.401,-77.418,179.762,14.875,151.169
C03122=1105.284,286.648,-77.447,179.766,14.876,151.168
C03123=1105.290,286.897,-77.477,179.769,14.877,151.167
C03124=1105.295,287.145,-77.506,179.773,14.878,151.167
C03125=1105.301,287.393,-77.537,179.777,14.879,151.166
C03126=1105.307,287.641,-77.566,179.781,14.880,151.165
C03127=1105.313,287.890,-77.595,179.784,14.881,151.165
C03128=1105.318,288.138,-77.625,179.788,14.881,151.164
C03129=1105.324,288.386,-77.655,179.792,14.882,151.164
C03130=1105.330,288.634,-77.684,179.795,14.883,151.163
C03131=1105.336,288.882,-77.714,179.800,14.884,151.162
C03132=1105.344,289.247,-77.758,179.805,14.885,151.162
C03133=1105.353,289.612,-77.802,179.810,14.887,151.161
C03134=1105.361,289.978,-77.845,179.816,14.888,151.160
C03135=1105.369,290.343,-77.889,179.821,14.889,151.159
C03136=1105.375,290.592,-77.919,179.824,14.890,151.158
C03137=1105.380,290.840,-77.949,179.829,14.891,151.158
C03138=1105.386,291.087,-77.978,179.832,14.892,151.157
C03139=1105.392,291.335,-78.008,179.836,14.893,151.156
C03140=1105.397,291.583,-78.038,179.839,14.894,151.156
C03141=1105.403,291.832,-78.068,179.844,14.895,151.155
C03142=1105.409,292.080,-78.098,179.847,14.895,151.155
C03143=1105.414,292.328,-78.127,179.851,14.897,151.154
C03144=1105.420,292.576,-78.158,179.854,14.897,151.154
C03145=1105.426,292.824,-78.187,179.858,14.898,151.153
C03146=1105.431,293.072,-78.218,179.862,14.899,151.152
C03147=1105.437,293.321,-78.247,179.866,14.900,151.152
C03148=1105.443,293.568,-78.278,179.869,14.901,151.151
C03149=1105.448,293.817,-78.307,179.872,14.902,151.151
C03150=1105.454,294.065,-78.338,179.876,14.903,151.150
C03151=1105.460,294.313,-78.367,179.880,14.904,151.149
C03152=1105.465,294.561,-78.398,179.884,14.905,151.149
C03153=1105.471,294.809,-78.428,179.887,14.906,151.148
C03154=1105.477,295.057,-78.458,179.891,14.907,151.148
C03155=1105.483,295.305,-78.488,179.895,14.908,151.147
C03156=1105.488,295.553,-78.518,179.898,14.909,151.147
C03157=1105.494,295.801,-78.548,179.902,14.910,151.146
C03158=1105.500,296.049,-78.578,179.906,14.911,151.145
C03159=1105.505,296.297,-78.609,179.909,14.912,151.145
C03160=1105.511,296.545,-78.638,179.913,14.913,151.144
C03161=1105.516,296.793,-78.669,179.917,14.914,151.144
C03162=1105.522,297.041,-78.700,179.920,14.915,151.143
C03163=1105.527,297.290,-78.729,179.924,14.916,151.143
C03164=1105.533,297.538,-78.760,179.928,14.917,151.142
C03165=1105.539,297.785,-78.790,179.931,14.918,151.142
C03166=1105.545,298.034,-78.821,179.935,14.920,151.141
C03167=1105.551,298.282,-78.851,179.939,14.920,151.140
C03168=1105.556,298.530,-78.881,179.942,14.921,151.140
C03169=1105.562,298.778,-78.912,179.946,14.923,151.139
C03170=1105.568,299.026,-78.942,179.950,14.924,151.139
C03171=1105.573,299.274,-78.973,179.954,14.925,151.138
C03172=1105.579,299.522,-79.003,179.957,14.926,151.138
C03173=1105.584,299.770,-79.034,179.961,14.927,151.137
C03174=1105.590,300.018,-79.063,179.964,14.928,151.137
C03175=1105.595,300.266,-79.094,179.968,14.930,151.136
C03176=1105.601,300.514,-79.125,179.971,14.930,151.136
C03177=1105.607,300.762,-79.155,179.975,14.932,151.135
C03178=1105.612,301.010,-79.186,179.979,14.933,151.135
C03179=1105.618,301.258,-79.216,179.982,14.934,151.134
C03180=1105.623,301.506,-79.247,179.986,14.936,151.134
C03181=1105.628,301.754,-79.278,179.989,14.937,151.133
C03182=1105.634,302.002,-79.308,179.993,14.938,151.133
C03183=1105.640,302.251,-79.339,179.996,14.939,151.132
C03184=1105.648,302.630,-79.386,-179.997,14.941,151.131
C03185=1105.657,303.009,-79.432,-179.992,14.942,151.131
C03186=1105.666,303.387,-79.479,-179.986,14.945,151.130
C03187=1105.674,303.767,-79.526,-179.981,14.946,151.129
C03188=1105.680,304.015,-79.557,-179.977,14.948,151.129
C03189=1105.685,304.263,-79.588,-179.974,14.948,151.128
C03190=1105.691,304.511,-79.618,-179.970,14.950,151.128
C03191=1105.697,304.759,-79.649,-179.966,14.951,151.127
C03192=1105.702,305.007,-79.680,-179.963,14.952,151.127
C03193=1105.708,305.254,-79.711,-179.959,14.954,151.126
C03194=1105.714,305.503,-79.742,-179.956,14.955,151.126
C03195=1105.720,305.751,-79.772,-179.952,14.956,151.125
C03196=1105.725,305.999,-79.803,-179.948,14.958,151.125
C03197=1105.731,306.246,-79.834,-179.945,14.958,151.124
C03198=1105.736,306.494,-79.865,-179.941,14.960,151.124
C03199=1105.742,306.743,-79.896,-179.938,14.961,151.123
C03200=1105.747,306.991,-79.927,-179.934,14.962,151.123
C03201=1105.754,307.238,-79.958,-179.930,14.964,151.122
C03202=1105.759,307.486,-79.989,-179.927,14.965,151.122
C03203=1105.765,307.735,-80.020,-179.923,14.967,151.121
C03204=1105.770,307.983,-80.051,-179.920,14.967,151.121
C03205=1105.776,308.230,-80.082,-179.916,14.969,151.120
C03206=1105.782,308.479,-80.113,-179.912,14.970,151.120
C03207=1105.788,308.726,-80.144,-179.909,14.971,151.119
C03208=1105.793,308.974,-80.175,-179.905,14.973,151.119
C03209=1105.799,309.222,-80.206,-179.901,14.974,151.118
C03210=1105.805,309.471,-80.238,-179.898,14.975,151.118
C03211=1105.810,309.719,-80.268,-179.894,14.977,151.117
C03212=1105.816,309.966,-80.300,-179.891,14.978,151.117
C03213=1105.822,310.215,-80.331,-179.887,14.979,151.116
C03214=1105.828,310.462,-80.362,-179.883,14.981,151.116
C03215=1105.833,310.710,-80.393,-179.880,14.982,151.115
C03216=1105.839,310.958,-80.425,-179.876,14.983,151.115
C03217=1105.845,311.206,-80.455,-179.873,14.985,151.115
C03218=1105.850,311.454,-80.487,-179.869,14.986,151.114
C03219=1105.857,311.702,-80.518,-179.866,14.988,151.114
C03220=1105.862,311.950,-80.549,-179.862,14.988,151.113
C03221=1105.868,312.198,-80.581,-179.858,14.990,151.113
C03222=1105.874,312.446,-80.612,-179.855,14.992,151.112
C03223=1105.879,312.693,-80.643,-179.852,14.993,151.112
C03224=1105.885,312.942,-80.675,-179.848,14.994,151.111
C03225=1105.891,313.189,-80.706,-179.844,14.996,151.111
C03226=1105.897,313.438,-80.737,-179.841,14.997,151.111
C03227=1105.902,313.686,-80.769,-179.837,14.998,151.110
C03228=1105.909,313.933,-80.800,-179.834,14.999,151.110
C03229=1105.914,314.182,-80.831,-179.830,15.001,151.109
C03230=1105.919,314.429,-80.863,-179.826,15.003,151.109
C03231=1105.925,314.677,-80.895,-179.823,15.004,151.108
C03232=1105.931,314.925,-80.925,-179.819,15.005,151.108
C03233=1105.937,315.173,-80.957,-179.816,15.007,151.107
C03234=1105.942,315.421,-80.989,-179.813,15.008,151.107
C03235=1105.948,315.669,-81.021,-179.809,15.010,151.107
C03236=1105.956,316.051,-81.068,-179.803,15.012,151.106
C03237=1105.965,316.433,-81.117,-179.798,15.014,151.105
C03238=1105.974,316.815,-81.166,-179.793,15.017,151.105
C03239=1105.982,317.196,-81.214,-179.787,15.019,151.104
C03240=1105.988,317.444,-81.246,-179.783,15.021,151.104
C03241=1105.994,317.691,-81.278,-179.780,15.022,151.103
C03242=1106.000,317.940,-81.310,-179.777,15.024,151.103
C03243=1106.004,318.188,-81.342,-179.773,15.026,151.103
C03244=1106.010,318.436,-81.374,-179.770,15.027,151.102
C03245=1106.016,318.683,-81.406,-179.766,15.029,151.102
C03246=1106.022,318.932,-81.437,-179.763,15.030,151.101
C03247=1106.027,319.180,-81.469,-179.759,15.032,151.101
C03248=1106.032,319.427,-81.501,-179.756,15.034,151.101
C03249=1106.038,319.675,-81.533,-179.752,15.035,151.100
C03250=1106.044,319.923,-81.564,-179.749,15.037,151.100
C03251=1106.050,320.171,-81.596,-179.746,15.038,151.100
C03252=1106.055,320.419,-81.628,-179.742,15.040,151.099
C03253=1106.061,320.667,-81.660,-179.738,15.042,151.099
C03254=1106.067,320.915,-81.692,-179.735,15.044,151.098
C03255=1106.072,321.162,-81.724,-179.732,15.045,151.098
C03256=1106.078,321.411,-81.756,-179.728,15.047,151.098
C03257=1106.083,321.659,-81.788,-179.724,15.048,151.097
C03258=1106.089,321.907,-81.820,-179.721,15.050,151.097
C03259=1106.094,322.154,-81.852,-179.718,15.051,151.097
C03260=1106.101,322.402,-81.884,-179.714,15.053,151.096
C03261=1106.106,322.649,-81.916,-179.711,15.055,151.096
C03262=1106.112,322.898,-81.948,-179.707,15.057,151.096
C03263=1106.117,323.145,-81.980,-179.704,15.058,151.095
C03264=1106.123,323.394,-82.012,-179.700,15.060,151.095
C03265=1106.129,323.642,-82.044,-179.697,15.062,151.095
C03266=1106.134,323.889,-82.076,-179.693,15.064,151.094
C03267=1106.140,324.137,-82.109,-179.690,15.065,151.094
C03268=1106.146,324.385,-82.141,-179.687,15.067,151.094
C03269=1106.151,324.633,-82.173,-179.683,15.069,151.093
C03270=1106.157,324.881,-82.205,-179.679,15.071,151.093
C03271=1106.163,325.128,-82.238,-179.676,15.072,151.093
C03272=1106.169,325.376,-82.270,-179.673,15.074,151.092
C03273=1106.175,325.624,-82.302,-179.669,15.076,151.092
C03274=1106.179,325.872,-82.334,-179.666,15.078,151.092
C03275=1106.186,326.120,-82.367,-179.662,15.080,151.091
C03276=1106.192,326.368,-82.399,-179.659,15.081,151.091
C03277=1106.197,326.616,-82.430,-179.656,15.083,151.091
C03278=1106.203,326.864,-82.464,-179.652,15.085,151.090
C03279=1106.209,327.112,-82.496,-179.648,15.087,151.090
C03280=1106.214,327.359,-82.527,-179.645,15.088,151.090
C03281=1106.220,327.607,-82.560,-179.642,15.090,151.089
C03282=1106.225,327.855,-82.593,-179.638,15.092,151.089
C03283=1106.232,328.103,-82.625,-179.635,15.094,151.089
C03284=1106.237,328.350,-82.657,-179.631,15.096,151.088
C03285=1106.243,328.598,-82.690,-179.628,15.097,151.088
C03286=1106.249,328.847,-82.722,-179.625,15.099,151.088
C03287=1106.255,329.094,-82.755,-179.621,15.101,151.088
C03288=1106.263,329.469,-82.803,-179.616,15.104,151.087
C03289=1106.272,329.843,-82.853,-179.611,15.106,151.087
C03290=1106.280,330.218,-82.903,-179.605,15.109,151.086
C03291=1106.289,330.593,-82.952,-179.601,15.112,151.086
C03292=1106.295,330.841,-82.984,-179.597,15.114,151.085
C03293=1106.301,331.088,-83.017,-179.594,15.116,151.085
C03294=1106.306,331.337,-83.049,-179.590,15.118,151.085
C03295=1106.313,331.585,-83.082,-179.586,15.120,151.085
C03296=1106.318,331.832,-83.115,-179.583,15.122,151.084
C03297=1106.324,332.080,-83.147,-179.580,15.123,151.084
C03298=1106.330,332.328,-83.180,-179.577,15.125,151.084
C03299=1106.336,332.575,-83.213,-179.573,15.127,151.083
C03300=1106.341,332.824,-83.246,-179.570,15.129,151.083
C03301=1106.346,333.071,-83.278,-179.566,15.131,151.083
C03302=1106.352,333.319,-83.312,-179.563,15.133,151.083
C03303=1106.358,333.567,-83.344,-179.560,15.136,151.083
C03304=1106.364,333.815,-83.377,-179.556,15.138,151.082
C03305=1106.369,334.062,-83.409,-179.553,15.140,151.082
C03306=1106.375,334.310,-83.443,-179.550,15.141,151.082
C03307=1106.380,334.558,-83.475,-179.547,15.144,151.082
C03308=1106.386,334.806,-83.508,-179.543,15.145,151.081
C03309=1106.392,335.054,-83.541,-179.540,15.148,151.081
C03310=1106.397,335.302,-83.575,-179.536,15.150,151.081
C03311=1106.403,335.548,-83.607,-179.533,15.152,151.081
C03312=1106.409,335.796,-83.640,-179.529,15.154,151.080
C03313=1106.414,336.045,-83.673,-179.526,15.156,151.080
C03314=1106.420,336.293,-83.706,-179.522,15.158,151.080
C03315=1106.426,336.540,-83.739,-179.519,15.161,151.080
C03316=1106.431,336.788,-83.772,-179.516,15.163,151.080
C03317=1106.438,337.036,-83.805,-179.512,15.165,151.079
C03318=1106.443,337.283,-83.838,-179.510,15.167,151.079
C03319=1106.448,337.531,-83.871,-179.506,15.168,151.079
C03320=1106.454,337.779,-83.904,-179.503,15.171,151.079
C03321=1106.460,338.027,-83.938,-179.499,15.173,151.078
C03322=1106.466,338.274,-83.971,-179.496,15.175,151.078
C03323=1106.472,338.522,-84.004,-179.493,15.177,151.078
C03324=1106.477,338.770,-84.037,-179.489,15.179,151.078
C03325=1106.483,339.018,-84.070,-179.486,15.182,151.078
C03326=1106.489,339.266,-84.104,-179.483,15.184,151.078
C03327=1106.493,339.513,-84.137,-179.480,15.186,151.077
C03328=1106.500,339.761,-84.169,-179.476,15.189,151.077
C03329=1106.505,340.008,-84.203,-179.473,15.191,151.077
C03330=1106.511,340.256,-84.236,-179.469,15.193,151.077
C03331=1106.517,340.504,-84.270,-179.466,15.195,151.077
C03332=1106.522,340.752,-84.303,-179.463,15.198,151.077
C03333=1106.528,340.999,-84.337,-179.460,15.200,151.076
C03334=1106.533,341.247,-84.370,-179.456,15.202,151.076
C03335=1106.540,341.495,-84.403,-179.453,15.205,151.076
C03336=1106.545,341.743,-84.436,-179.450,15.207,151.076
C03337=1106.551,341.990,-84.470,-179.446,15.209,151.076
C03338=1106.557,342.238,-84.504,-179.443,15.211,151.076
C03339=1106.562,342.486,-84.537,-179.440,15.214,151.075
C03340=1106.570,342.854,-84.587,-179.435,15.217,151.075
C03341=1106.579,343.223,-84.637,-179.430,15.221,151.075
C03342=1106.588,343.592,-84.686,-179.425,15.224,151.075
C03343=1106.596,343.960,-84.736,-179.420,15.228,151.075
C03344=1106.601,344.208,-84.769,-179.417,15.230,151.075
C03345=1106.607,344.455,-84.803,-179.414,15.233,151.075
C03346=1106.613,344.703,-84.837,-179.411,15.235,151.074
C03347=1106.619,344.950,-84.871,-179.408,15.237,151.074
C03348=1106.624,345.198,-84.904,-179.404,15.240,151.074
C03349=1106.630,345.446,-84.937,-179.401,15.242,151.074
C03350=1106.636,345.693,-84.971,-179.398,15.244,151.074
C03351=1106.641,345.941,-85.005,-179.395,15.247,151.074
C03352=1106.648,346.189,-85.039,-179.392,15.249,151.074
C03353=1106.653,346.437,-85.073,-179.388,15.252,151.074
C03354=1106.659,346.684,-85.107,-179.384,15.255,151.074
C03355=1106.665,346.932,-85.140,-179.381,15.257,151.073
C03356=1106.670,347.180,-85.175,-179.378,15.260,151.073
C03357=1106.675,347.428,-85.208,-179.375,15.262,151.073
C03358=1106.681,347.675,-85.242,-179.372,15.264,151.073
C03359=1106.687,347.923,-85.275,-179.369,15.267,151.073
C03360=1106.692,348.170,-85.309,-179.366,15.270,151.073
C03361=1106.698,348.418,-85.343,-179.363,15.272,151.073
C03362=1106.704,348.665,-85.377,-179.359,15.275,151.073
C03363=1106.709,348.913,-85.411,-179.356,15.277,151.073
C03364=1106.715,349.161,-85.445,-179.353,15.280,151.073
C03365=1106.720,349.408,-85.479,-179.349,15.283,151.073
C03366=1106.726,349.655,-85.513,-179.346,15.285,151.073
C03367=1106.732,349.903,-85.546,-179.343,15.288,151.073
C03368=1106.738,350.152,-85.581,-179.340,15.290,151.073
C03369=1106.743,350.399,-85.615,-179.337,15.293,151.073
C03370=1106.749,350.647,-85.649,-179.334,15.296,151.073
C03371=1106.755,350.894,-85.683,-179.331,15.298,151.072
C03372=1106.760,351.142,-85.717,-179.328,15.301,151.072
C03373=1106.766,351.389,-85.751,-179.324,15.304,151.072
C03374=1106.771,351.637,-85.785,-179.321,15.306,151.072
C03375=1106.778,351.885,-85.819,-179.318,15.309,151.072
C03376=1106.783,352.132,-85.854,-179.315,15.311,151.072
C03377=1106.789,352.380,-85.888,-179.312,15.314,151.072
C03378=1106.795,352.627,-85.922,-179.309,15.317,151.072
C03379=1106.800,352.875,-85.957,-179.305,15.320,151.072
C03380=1106.805,353.122,-85.990,-179.302,15.323,151.072
C03381=1106.812,353.370,-86.024,-179.299,15.325,151.072
C03382=1106.817,353.618,-86.059,-179.296,15.328,151.072
C03383=1106.823,353.865,-86.093,-179.293,15.331,151.072
C03384=1106.829,354.113,-86.127,-179.290,15.333,151.072
C03385=1106.834,354.360,-86.162,-179.286,15.337,151.072
C03386=1106.840,354.607,-86.196,-179.283,15.339,151.072
C03387=1106.845,354.856,-86.231,-179.280,15.342,151.072
C03388=1106.851,355.103,-86.265,-179.277,15.345,151.072
C03389=1106.857,355.350,-86.299,-179.274,15.347,151.072
C03390=1106.862,355.598,-86.334,-179.271,15.351,151.072
C03391=1106.868,355.845,-86.368,-179.268,15.354,151.072
C03392=1106.876,356.216,-86.420,-179.263,15.358,151.073
C03393=1106.885,356.587,-86.471,-179.259,15.362,151.073
C03394=1106.893,356.958,-86.523,-179.254,15.367,151.073
C03395=1106.902,357.328,-86.575,-179.249,15.371,151.073
C03396=1106.908,357.576,-86.609,-179.246,15.373,151.073
C03397=1106.913,357.823,-86.643,-179.243,15.377,151.073
C03398=1106.918,358.071,-86.678,-179.240,15.379,151.073
C03399=1106.925,358.319,-86.712,-179.237,15.383,151.073
C03400=1106.930,358.566,-86.747,-179.234,15.385,151.073
C03401=1106.936,358.813,-86.782,-179.230,15.389,151.073
C03402=1106.942,359.061,-86.817,-179.228,15.391,151.073
C03403=1106.948,359.309,-86.851,-179.225,15.394,151.073
C03404=1106.953,359.556,-86.885,-179.222,15.397,151.073
C03405=1106.958,359.803,-86.921,-179.218,15.401,151.073
C03406=1106.965,360.051,-86.955,-179.215,15.403,151.073
C03407=1106.970,360.299,-86.990,-179.212,15.406,151.074
C03408=1106.976,360.545,-87.025,-179.210,15.409,151.074
C03409=1106.982,360.794,-87.060,-179.206,15.413,151.074
C03410=1106.987,361.041,-87.094,-179.204,15.416,151.074
C03411=1106.993,361.288,-87.129,-179.201,15.419,151.074
C03412=1106.999,361.536,-87.164,-179.197,15.422,151.074
C03413=1107.004,361.784,-87.199,-179.194,15.425,151.074
C03414=1107.010,362.030,-87.233,-179.191,15.428,151.074
C03415=1107.015,362.278,-87.268,-179.189,15.431,151.075
C03416=1107.021,362.526,-87.304,-179.185,15.434,151.075
C03417=1107.026,362.773,-87.338,-179.182,15.437,151.075
C03418=1107.033,363.020,-87.373,-179.180,15.440,151.075
C03419=1107.038,363.268,-87.408,-179.176,15.444,151.075
C03420=1107.043,363.516,-87.443,-179.174,15.447,151.075
C03421=1107.050,363.763,-87.478,-179.171,15.450,151.075
C03422=1107.056,364.010,-87.513,-179.167,15.454,151.075
C03423=1107.061,364.258,-87.548,-179.165,15.457,151.076
C03424=1107.067,364.505,-87.584,-179.162,15.459,151.076
C03425=1107.072,364.753,-87.618,-179.158,15.463,151.076
C03426=1107.078,365.000,-87.653,-179.156,15.466,151.076
C03427=1107.084,365.248,-87.688,-179.153,15.469,151.076
C03428=1107.089,365.495,-87.724,-179.149,15.473,151.076
C03429=1107.095,365.743,-87.759,-179.147,15.476,151.077
C03430=1107.100,365.990,-87.794,-179.144,15.479,151.077
C03431=1107.107,366.237,-87.829,-179.141,15.483,151.077
C03432=1107.113,366.485,-87.864,-179.138,15.486,151.077
C03433=1107.118,366.732,-87.899,-179.135,15.490,151.077
C03434=1107.123,366.979,-87.934,-179.132,15.493,151.078
C03435=1107.129,367.227,-87.970,-179.130,15.496,151.078
C03436=1107.134,367.474,-88.005,-179.126,15.500,151.078
C03437=1107.140,367.722,-88.041,-179.124,15.503,151.078
C03438=1107.146,367.969,-88.076,-179.120,15.507,151.079
C03439=1107.151,368.216,-88.111,-179.118,15.510,151.079
C03440=1107.157,368.464,-88.146,-179.115,15.513,151.079
C03441=1107.162,368.711,-88.182,-179.112,15.517,151.079
C03442=1107.168,368.959,-88.217,-179.109,15.520,151.080
C03443=1107.174,369.206,-88.253,-179.106,15.524,151.080
C03444=1107.183,369.592,-88.308,-179.101,15.529,151.080
C03445=1107.192,369.977,-88.363,-179.098,15.534,151.081
C03446=1107.201,370.363,-88.418,-179.093,15.540,151.081
C03447=1107.209,370.748,-88.473,-179.089,15.545,151.081
C03448=1107.215,370.995,-88.509,-179.085,15.549,151.082
C03449=1107.221,371.243,-88.545,-179.083,15.553,151.082
C03450=1107.226,371.490,-88.580,-179.080,15.556,151.082
C03451=1107.232,371.738,-88.616,-179.077,15.560,151.082
C03452=1107.238,371.985,-88.651,-179.074,15.564,151.083
C03453=1107.244,372.232,-88.687,-179.071,15.567,151.083
C03454=1107.249,372.479,-88.722,-179.068,15.571,151.083
C03455=1107.254,372.727,-88.758,-179.066,15.574,151.084
C03456=1107.260,372.974,-88.794,-179.063,15.578,151.084
C03457=1107.266,373.221,-88.830,-179.060,15.581,151.084
C03458=1107.272,373.468,-88.866,-179.058,15.585,151.085
C03459=1107.278,373.716,-88.901,-179.055,15.589,151.085
C03460=1107.283,373.963,-88.937,-179.052,15.592,151.085
C03461=1107.289,374.211,-88.972,-179.049,15.596,151.085
C03462=1107.295,374.458,-89.008,-179.046,15.599,151.086
C03463=1107.300,374.706,-89.044,-179.043,15.604,151.086
C03464=1107.306,374.953,-89.081,-179.041,15.607,151.086
C03465=1107.312,375.200,-89.116,-179.038,15.611,151.087
C03466=1107.318,375.447,-89.152,-179.035,15.615,151.087
C03467=1107.322,375.695,-89.188,-179.033,15.619,151.088
C03468=1107.328,375.942,-89.223,-179.030,15.623,151.088
C03469=1107.334,376.189,-89.259,-179.027,15.627,151.088
C03470=1107.340,376.436,-89.295,-179.024,15.631,151.089
C03471=1107.345,376.683,-89.331,-179.022,15.634,151.089
C03472=1107.351,376.931,-89.368,-179.019,15.638,151.090
C03473=1107.357,377.178,-89.403,-179.017,15.642,151.090
C03474=1107.362,377.425,-89.439,-179.013,15.646,151.090
C03475=1107.368,377.673,-89.476,-179.010,15.650,151.091
C03476=1107.374,377.920,-89.511,-179.008,15.654,151.091
C03477=1107.379,378.168,-89.547,-179.005,15.658,151.091
C03478=1107.385,378.414,-89.583,-179.003,15.661,151.092
C03479=1107.391,378.662,-89.619,-179.000,15.666,151.092
C03480=1107.396,378.909,-89.656,-178.997,15.670,151.093
C03481=1107.402,379.156,-89.692,-178.995,15.674,151.093
C03482=1107.407,379.403,-89.729,-178.992,15.678,151.093
C03483=1107.413,379.650,-89.764,-178.990,15.682,151.094
C03484=1107.419,379.898,-89.800,-178.987,15.686,151.094
C03485=1107.424,380.145,-89.837,-178.983,15.690,151.095
C03486=1107.430,380.392,-89.873,-178.981,15.694,151.095
C03487=1107.435,380.640,-89.909,-178.978,15.698,151.096
C03488=1107.442,380.887,-89.946,-178.976,15.702,151.096
C03489=1107.447,381.134,-89.981,-178.973,15.706,151.097
C03490=1107.453,381.381,-90.018,-178.970,15.710,151.097
C03491=1107.459,381.629,-90.054,-178.968,15.714,151.098
C03492=1107.464,381.875,-90.090,-178.965,15.718,151.098
C03493=1107.470,382.122,-90.127,-178.962,15.723,151.099
C03494=1107.475,382.370,-90.163,-178.960,15.726,151.099
C03495=1107.482,382.617,-90.200,-178.957,15.731,151.099
C03496=1107.491,383.029,-90.260,-178.953,15.738,151.100
C03497=1107.500,383.441,-90.322,-178.948,15.745,151.101
C03498=1107.509,383.853,-90.381,-178.945,15.752,151.102
C03499=1107.519,384.266,-90.443,-178.941,15.759,151.103
C03500=1107.525,384.513,-90.479,-178.938,15.764,151.103
C03501=1107.530,384.760,-90.516,-178.935,15.768,151.104
C03502=1107.536,385.008,-90.552,-178.933,15.772,151.105
C03503=1107.541,385.254,-90.589,-178.930,15.777,151.105
C03504=1107.547,385.502,-90.626,-178.928,15.781,151.106
C03505=1107.553,385.749,-90.662,-178.925,15.786,151.106
C03506=1107.558,385.995,-90.699,-178.923,15.790,151.107
C03507=1107.564,386.243,-90.736,-178.920,15.794,151.107
C03508=1107.570,386.490,-90.772,-178.917,15.799,151.108
C03509=1107.576,386.737,-90.809,-178.915,15.804,151.109
C03510=1107.580,386.984,-90.845,-178.912,15.808,151.109
C03511=1107.586,387.232,-90.882,-178.910,15.812,151.110
C03512=1107.592,387.479,-90.919,-178.907,15.817,151.110
C03513=1107.598,387.726,-90.956,-178.905,15.821,151.111
C03514=1107.603,387.973,-90.992,-178.902,15.826,151.111
C03515=1107.609,388.220,-91.029,-178.900,15.830,151.112
C03516=1107.615,388.467,-91.066,-178.898,15.835,151.113
C03517=1107.620,388.715,-91.103,-178.895,15.839,151.113
C03518=1107.626,388.962,-91.140,-178.892,15.844,151.114
C03519=1107.632,389.208,-91.177,-178.890,15.849,151.115
C03520=1107.638,389.455,-91.214,-178.887,15.854,151.115
C03521=1107.643,389.702,-91.251,-178.885,15.858,151.116
C03522=1107.649,389.950,-91.288,-178.883,15.863,151.117
C03523=1107.654,390.197,-91.325,-178.880,15.867,151.117
C03524=1107.661,390.444,-91.361,-178.878,15.872,151.118
C03525=1107.666,390.691,-91.398,-178.875,15.876,151.118
C03526=1107.671,390.938,-91.435,-178.872,15.881,151.119
C03527=1107.677,391.185,-91.473,-178.871,15.886,151.120
C03528=1107.683,391.432,-91.510,-178.868,15.891,151.120
C03529=1107.689,391.679,-91.546,-178.865,15.895,151.121
C03530=1107.695,391.927,-91.583,-178.863,15.900,151.122
C03531=1107.701,392.173,-91.621,-178.861,15.905,151.122
C03532=1107.706,392.421,-91.658,-178.858,15.910,151.123
C03533=1107.712,392.668,-91.695,-178.856,15.915,151.124
C03534=1107.717,392.915,-91.732,-178.854,15.919,151.125
C03535=1107.723,393.162,-91.770,-178.851,15.924,151.125
C03536=1107.728,393.409,-91.807,-178.849,15.929,151.126
C03537=1107.734,393.656,-91.844,-178.847,15.934,151.127
C03538=1107.740,393.903,-91.882,-178.844,15.939,151.128
C03539=1107.746,394.150,-91.919,-178.842,15.944,151.128
C03540=1107.751,394.398,-91.956,-178.839,15.949,151.129
C03541=1107.757,394.645,-91.993,-178.837,15.954,151.130
C03542=1107.763,394.892,-92.030,-178.835,15.959,151.131
C03543=1107.768,395.139,-92.067,-178.832,15.964,151.131
C03544=1107.774,395.386,-92.105,-178.830,15.969,151.132
C03545=1107.780,395.633,-92.142,-178.829,15.973,151.133
C03546=1107.786,395.880,-92.180,-178.826,15.978,151.134
C03547=1107.791,396.128,-92.217,-178.824,15.984,151.135
C03548=1107.796,396.339,-92.250,-178.821,15.989,151.135
C03549=1107.801,396.551,-92.281,-178.820,15.993,151.136
C03550=1107.805,396.764,-92.314,-178.818,15.997,151.137
C03551=1107.810,396.975,-92.346,-178.816,16.001,151.137
C03552=1107.815,397.188,-92.378,-178.814,16.006,151.138
C03553=1107.820,397.400,-92.411,-178.812,16.010,151.139
C03554=1107.825,397.612,-92.442,-178.810,16.015,151.139
C03555=1107.829,397.824,-92.475,-178.808,16.020,151.140
C03556=1107.835,398.071,-92.512,-178.806,16.025,151.141
C03557=1107.841,398.318,-92.550,-178.804,16.030,151.142
C03558=1107.847,398.565,-92.587,-178.801,16.035,151.143
C03559=1107.852,398.812,-92.625,-178.799,16.041,151.144
C03560=1107.858,399.059,-92.663,-178.797,16.046,151.145
C03561=1107.863,399.307,-92.700,-178.795,16.051,151.145
C03562=1107.869,399.553,-92.738,-178.793,16.057,151.146
C03563=1107.875,399.800,-92.776,-178.791,16.062,151.147
C03564=1107.880,400.048,-92.813,-178.788,16.067,151.148
C03565=1107.886,400.294,-92.851,-178.786,16.072,151.149
C03566=1107.892,400.541,-92.889,-178.784,16.078,151.150
C03567=1107.897,400.789,-92.928,-178.782,16.083,151.151
C03568=1107.903,401.036,-92.965,-178.780,16.089,151.152
C03569=1107.909,401.283,-93.002,-178.778,16.094,151.153
C03570=1107.914,401.530,-93.041,-178.776,16.100,151.154
C03571=1107.920,401.777,-93.078,-178.773,16.105,151.155
C03572=1107.926,402.024,-93.116,-178.771,16.111,151.155
C03573=1107.931,402.271,-93.154,-178.769,16.116,151.156
C03574=1107.937,402.518,-93.192,-178.767,16.122,151.157
C03575=1107.942,402.765,-93.230,-178.765,16.127,151.158
C03576=1107.948,403.012,-93.268,-178.763,16.133,151.159
C03577=1107.954,403.259,-93.306,-178.761,16.138,151.160
C03578=1107.959,403.506,-93.344,-178.758,16.145,151.161
C03579=1107.965,403.753,-93.382,-178.757,16.150,151.162
C03580=1107.971,404.000,-93.420,-178.755,16.156,151.163
C03581=1107.976,404.247,-93.458,-178.753,16.161,151.164
C03582=1107.981,404.495,-93.496,-178.751,16.167,151.165
C03583=1107.988,404.742,-93.534,-178.748,16.173,151.166
C03584=1107.993,404.989,-93.572,-178.746,16.179,151.167
C03585=1107.999,405.236,-93.610,-178.744,16.184,151.168
C03586=1108.004,405.482,-93.649,-178.742,16.190,151.169
C03587=1108.010,405.729,-93.687,-178.741,16.196,151.170
C03588=1108.015,405.976,-93.725,-178.738,16.202,151.172
C03589=1108.022,406.223,-93.763,-178.736,16.208,151.173
C03590=1108.027,406.471,-93.802,-178.734,16.214,151.174
C03591=1108.033,406.717,-93.839,-178.732,16.220,151.175
C03592=1108.038,406.964,-93.878,-178.730,16.226,151.176
C03593=1108.043,407.211,-93.916,-178.728,16.232,151.177
C03594=1108.050,407.459,-93.954,-178.726,16.237,151.178
C03595=1108.055,407.706,-93.992,-178.724,16.244,151.179
C03596=1108.061,407.952,-94.031,-178.722,16.250,151.180
C03597=1108.066,408.199,-94.069,-178.721,16.256,151.182
C03598=1108.072,408.447,-94.108,-178.718,16.262,151.183
C03599=1108.078,408.694,-94.146,-178.716,16.268,151.184
C03600=1108.083,408.940,-94.185,-178.715,16.274,151.185
C03601=1108.089,409.187,-94.223,-178.712,16.280,151.186
C03602=1108.094,409.434,-94.262,-178.711,16.286,151.187
C03603=1108.100,409.682,-94.300,-178.708,16.293,151.188
C03604=1108.105,409.893,-94.332,-178.707,16.298,151.189
C03605=1108.110,410.104,-94.366,-178.705,16.304,151.190
C03606=1108.115,410.317,-94.399,-178.703,16.309,151.191
C03607=1108.120,410.529,-94.432,-178.702,16.314,151.192
C03608=1108.124,410.741,-94.466,-178.700,16.320,151.194
C03609=1108.129,410.953,-94.499,-178.699,16.325,151.195
C03610=1108.133,411.164,-94.532,-178.697,16.331,151.196
C03611=1108.138,411.376,-94.565,-178.695,16.336,151.197
C03612=1108.144,411.623,-94.603,-178.694,16.343,151.198
C03613=1108.150,411.870,-94.642,-178.692,16.349,151.199
C03614=1108.155,412.117,-94.680,-178.690,16.355,151.200
C03615=1108.161,412.364,-94.720,-178.688,16.362,151.202
C03616=1108.166,412.611,-94.758,-178.686,16.368,151.203
C03617=1108.172,412.858,-94.797,-178.684,16.375,151.204
C03618=1108.178,413.105,-94.835,-178.683,16.382,151.205
C03619=1108.184,413.352,-94.875,-178.680,16.388,151.207
C03620=1108.189,413.599,-94.913,-178.679,16.395,151.208
C03621=1108.194,413.845,-94.952,-178.677,16.401,151.209
C03622=1108.200,414.093,-94.991,-178.675,16.408,151.211
C03623=1108.206,414.339,-95.030,-178.673,16.415,151.212
C03624=1108.212,414.586,-95.069,-178.672,16.421,151.213
C03625=1108.218,414.833,-95.107,-178.670,16.428,151.215
C03626=1108.223,415.080,-95.146,-178.668,16.434,151.216
C03627=1108.229,415.327,-95.185,-178.666,16.441,151.217
C03628=1108.234,415.574,-95.224,-178.664,16.448,151.219
C03629=1108.240,415.820,-95.263,-178.663,16.455,151.220
C03630=1108.246,416.067,-95.302,-178.661,16.462,151.221
C03631=1108.251,416.314,-95.341,-178.660,16.468,151.223
C03632=1108.257,416.562,-95.380,-178.657,16.475,151.224
